// TIA Portal V17 export
// export: Created 2024-06-14T09:52:20.614085Z, ExportSetting WithDefaults, DisplayName Totally Integrated Automation Portal, DisplayVersion V17, DisplayName TIA Portal Openness, DisplayVersion V17, DisplayName TIA Portal Version Control Interface, DisplayVersion V17, DisplayName Simotion SCOUT TIA, DisplayVersion 5.4.3.0, DisplayName SINAMICS Startdrive Advanced, DisplayVersion V17 SP1 Update 1, DisplayName SINAMICS Startdrive G110M, G120, G120C, G120D, G120P, G115D, DisplayVersion V17 SP1 Update 1, DisplayName SINAMICS Startdrive G130, G150, S120, S150, SINAMICS MV, S210, DisplayVersion V17 SP1 Update 1, DisplayName STEP 7 Professional, DisplayVersion V17, DisplayName STEP 7 Safety, DisplayVersion V17, DisplayName WinCC Professional, DisplayVersion V17
FUNCTION_BLOCK "FILLING_FB_L2"   // FB12, LAD
{ S7_Optimized_Access := 'TRUE' }
VERSION : 0.1
// stored: AutoNumber false, IsIECCheckEnabled false, IsRetainMemResEnabled false, MemoryReserve 100, SetENOAutomatically false, UDAEnableTagReadback false
   VAR_INPUT
      CYCLE_START : Bool;
      CYCLE_RESET : Bool;
      CYL_STOPPER : Bool;
      CYL_SENSOR1 : Bool;
      CYL_SENSOR2 : Bool;
      CYL_SENSOR3 : Bool;
      CYL_SENSOR4 : Bool;
      CYL_SENSOR5 : Bool;
      CYL_SENSOR6 : Bool;
      "DOWN CONVEYOR" : Bool;
      "SENSING TIME" : DInt;
      ENABLE_CYLINDER { ExternalAccessible := 'False'; ExternalVisible := 'False'; ExternalWritable := 'False'} : Array[1..6] of Bool;
      ENABLED_CYLINDER { ExternalAccessible := 'False'; ExternalVisible := 'False'; ExternalWritable := 'False'} : Int;
      GUN_DELAY_TIME : DInt;
      FILL_SEQ_STARTED : Array[1..6] of Bool;
      FILLING_DONE : Array[1..6] of Bool;
   END_VAR
   VAR_OUTPUT
      STOPPER : Bool;
      "LIFT TABLE1" : Bool;
      "LIFT TABLE2" : Bool;
      "LIFT TABLE3" : Bool;
      "LIFT TABLE4" : Bool;
      "LIFT TABLE5" : Bool;
      "LIFT TABLE6" : Bool;
      GUN_DOWN1 : Bool;
      GUN_DOWN2 : Bool;
      GUN_DOWN3 : Bool;
      GUN_DOWN4 : Bool;
      GUN_DOWN5 : Bool;
      GUN_DOWN6 : Bool;
      CYCLE_RUNNING : Bool;
      FILL_STT_SEQ1 : Bool;
      FILL_STT_SEQ2 : Bool;
      FILL_STT_SEQ3 : Bool;
      FILL_STT_SEQ4 : Bool;
      FILL_STT_SEQ5 : Bool;
      FILL_STT_SEQ6 : Bool;
      FILLING_SEQ_DONE : Bool;
      ALL_STATION_DISABLED : Bool;
   END_VAR
   VAR
      "FIRST SCAN BIT" : Bool;
      CYCLE_OK : Bool;
      CYCLE_RESTART : Bool;
      "COUNTER RESET" : Bool;
      FIRST_CYCLE : Bool;
      "CYL COUNT  VALUE" : Int;
      "PLUS BIT" : Array[1..50] of Bool;
      "GUN DOWN" : Bool;
   END_VAR
   VAR RETAIN
      TILLTING_TIME { S7_SetPoint := 'True'} : DInt;
      M1_DECLAMP_TIME : DInt;
      CYL_COUNTER_S1 { S7_SetPoint := 'True'} : CTU_INT;
      CYL_COUNTER_S2 { S7_SetPoint := 'True'} : CTU_INT;
      CYL_COUNTER_S3 { S7_SetPoint := 'True'} : CTU_INT;
      CYL_COUNTER_S4 { S7_SetPoint := 'True'} : CTU_INT;
      CYL_COUNTER_S5 { S7_SetPoint := 'True'} : CTU_INT;
      CYL_COUNTER_S6 { S7_SetPoint := 'True'} : CTU_INT;
      CYL_COUNTER_S11 { S7_SetPoint := 'True'} : CTU_INT;
      CYL_COUNT_CONT_S1 { S7_SetPoint := 'True'} : CTU_INT;
      CYL_COUNT_CONT_S2 { S7_SetPoint := 'True'} : CTU_INT;
      CYL_COUNT_CONT_S3 { S7_SetPoint := 'True'} : CTU_INT;
      CYL_COUNT_CONT_S4 { S7_SetPoint := 'True'} : CTU_INT;
      CYL_COUNT_CONT_S5 { S7_SetPoint := 'True'} : CTU_INT;
      CYL_COUNT_CONT_S6 { S7_SetPoint := 'True'} : CTU_INT;
      "STOPPER COUNTER" { S7_SetPoint := 'True'} : CTU_INT;
   END_VAR
   VAR
      CYL_STAB_S1 { S7_SetPoint := 'True'} : TON_TIME;
      CYL_STAB_S2 { S7_SetPoint := 'True'} : TON_TIME;
      CYL_STAB_S3 { S7_SetPoint := 'True'} : TON_TIME;
      CYL_STAB_S4 { S7_SetPoint := 'True'} : TON_TIME;
      CYL_STAB_S5 { S7_SetPoint := 'True'} : TON_TIME;
      CYL_STAB_S6 { S7_SetPoint := 'True'} : TON_TIME;
      CYCLE_RST_OFF { S7_SetPoint := 'True'} : TOF_TIME;
      CYCLE_RST_ON { S7_SetPoint := 'True'} : TON_TIME;
      DECLAMP_MUL : DInt;
      DECLAMP_ADD : DInt;
      "CYL STOPPER" : Bool;
      STOP_DLY { S7_SetPoint := 'True'} : TON_TIME;
      Disable_Stations { S7_SetPoint := 'True'} : "Disable";
      First_Cylinder : Array[1..6] of Int;
      Disab_Total_Cyl : Int;
      GUN_DOWN_FBK : Bool;
      GUN_DOWN_FBK_T { S7_SetPoint := 'True'} : TON_TIME;
      AUTO_RESTART : Bool;
      GUN_DOWN_1 { S7_SetPoint := 'True'} : TON_TIME;
      GUN_DOWN_2 { S7_SetPoint := 'True'} : TON_TIME;
      GUN_DOWN_3 { S7_SetPoint := 'True'} : TON_TIME;
      GUN_DOWN_4 { S7_SetPoint := 'True'} : TON_TIME;
      GUN_DOWN_5 { S7_SetPoint := 'True'} : TON_TIME;
      GUN_DOWN_6 { S7_SetPoint := 'True'} : TON_TIME;
      FILL_STT_1 { S7_SetPoint := 'True'} : TON_TIME;
      FILL_STT_2 { S7_SetPoint := 'True'} : TON_TIME;
      FILL_STT_3 { S7_SetPoint := 'True'} : TON_TIME;
      FILL_STT_4 { S7_SetPoint := 'True'} : TON_TIME;
      FILL_STT_5 { S7_SetPoint := 'True'} : TON_TIME;
      FILL_STT_6 { S7_SetPoint := 'True'} : TON_TIME;
      ALL_FILL_DONE : Bool;
      ALL_GUN_UP : Bool;
      AUTO_CYCLE { S7_SetPoint := 'True'} : TON_TIME;
      AUTO { S7_SetPoint := 'True'} : Bool;
      MANUAL { S7_SetPoint := 'True'} : Bool;
      Man_Gun_down_1 : Bool;
      Man_Gun_down_2 : Bool;
      Man_Gun_down_3 : Bool;
      Man_Gun_down_4 : Bool;
      Man_Gun_down_5 : Bool;
      Man_Gun_down_6 : Bool;
      Man_Lift_up_1 : Bool;
      Man_Lift_up_2 : Bool;
      Man_Lift_up_3 : Bool;
      Man_Lift_up_4 : Bool;
      Man_Lift_up_5 : Bool;
      Man_Lift_up_6 : Bool;
      trig : Array[0..50] of Bool;
      "trig count" : Array[0..10] of TON_TIME;
      delay : Time;
   END_VAR
   VAR_TEMP   // added for the SCL form of the ladder/FBD networks
      _w1 : Bool;
      _w2 : Bool;
      _w3 : Bool;
      _w4 : Bool;
      _w5 : Bool;
      _w6 : Bool;
      _w7 : Bool;
      _w8 : Bool;
      _w9 : Bool;
      _w10 : Bool;
      _w11 : Bool;
      _w12 : Bool;
      _w13 : Bool;
      _w14 : Bool;
      _w15 : Bool;
      _w16 : Bool;
      _w17 : Bool;
      _w18 : Bool;
      _w19 : Bool;
      _w20 : Bool;
      _w21 : Bool;
      _w22 : Bool;
      _w23 : Bool;
      _w24 : Bool;
      _w25 : Bool;
      _w26 : Bool;
      _w27 : Bool;
      _w28 : Bool;
      _w29 : Bool;
      _w30 : Bool;
      _w31 : Bool;
   END_VAR
BEGIN

REGION Network 2: CYCLE START / POWER RESET OFF
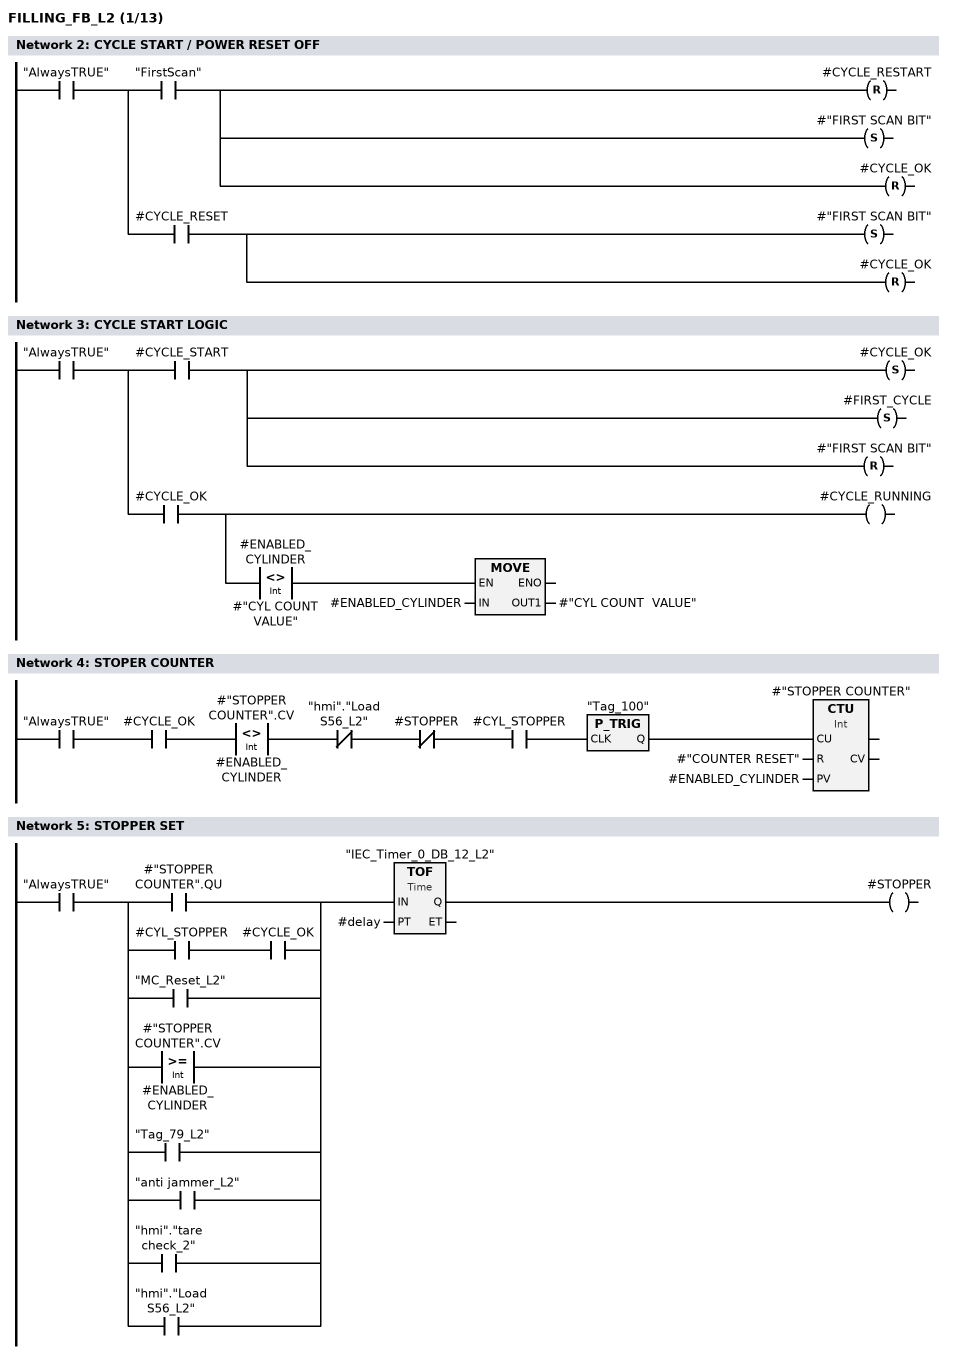
   RUNG wire#powerrail
      Contact( "AlwaysTRUE" )
      wire#w1
      Contact( "FirstScan" )
      wire#w2
      R_Coil( #CYCLE_RESTART )
   END_RUNG
   RUNG wire#w2
      S_Coil( #"FIRST SCAN BIT" )
   END_RUNG
   RUNG wire#w2
      R_Coil( #CYCLE_OK )
   END_RUNG
   RUNG wire#w1
      Contact( #CYCLE_RESET )
      wire#w3
      S_Coil( #"FIRST SCAN BIT" )
   END_RUNG
   RUNG wire#w3
      R_Coil( #CYCLE_OK )
   END_RUNG
   // the same network as SCL:
   IF "AlwaysTRUE" AND "FirstScan" THEN
       #CYCLE_RESTART := FALSE;
       #"FIRST SCAN BIT" := TRUE;
       #CYCLE_OK := FALSE;
   END_IF;
   IF "AlwaysTRUE" AND #CYCLE_RESET THEN
       #"FIRST SCAN BIT" := TRUE;
       #CYCLE_OK := FALSE;
   END_IF;
END_REGION

REGION Network 3: CYCLE START LOGIC
   RUNG wire#powerrail
      Contact( "AlwaysTRUE" )
      wire#w1
      Contact( #CYCLE_START )
      wire#w2
      S_Coil( #CYCLE_OK )
   END_RUNG
   RUNG wire#w2
      S_Coil( #FIRST_CYCLE )
   END_RUNG
   RUNG wire#w2
      R_Coil( #"FIRST SCAN BIT" )
   END_RUNG
   RUNG wire#w1
      Contact( #CYCLE_OK )
      wire#w3
      Coil( #CYCLE_RUNNING )
   END_RUNG
   RUNG wire#w3
      { S7_Templates := "SrcType := Int" } NE_Contact(in1 := #ENABLED_CYLINDER, in2 := #"CYL COUNT  VALUE")
      Move(in := #ENABLED_CYLINDER, out1 => #"CYL COUNT  VALUE")
   END_RUNG
   // the same network as SCL:
   IF "AlwaysTRUE" AND #CYCLE_START THEN
       #CYCLE_OK := TRUE;
       #FIRST_CYCLE := TRUE;
       #"FIRST SCAN BIT" := FALSE;
   END_IF;
   #CYCLE_RUNNING := "AlwaysTRUE" AND #CYCLE_OK;
   IF #CYCLE_RUNNING AND (#ENABLED_CYLINDER <> #"CYL COUNT  VALUE") THEN
       #"CYL COUNT  VALUE" := #ENABLED_CYLINDER;
   END_IF;
END_REGION

REGION Network 4: STOPER COUNTER
   RUNG wire#powerrail
      Contact( "AlwaysTRUE" )
      Contact( #CYCLE_OK )
      { S7_Templates := "SrcType := Int" } NE_Contact(in1 := #"STOPPER COUNTER".CV, in2 := #ENABLED_CYLINDER)
      I_Contact( "hmi"."Load S56_L2" )
      I_Contact( #STOPPER )
      Contact( #CYL_STOPPER )
      P_Trig( "Tag_100" )
      { S7_Templates := "value_type := Int" } #"STOPPER COUNTER".CTU(r := #"COUNTER RESET", pv := #ENABLED_CYLINDER, cv =>)
   END_RUNG
   // the same network as SCL:
   #_w1 := "AlwaysTRUE" AND #CYCLE_OK AND (#"STOPPER COUNTER".CV <> #ENABLED_CYLINDER) AND NOT "hmi"."Load S56_L2" AND NOT #STOPPER AND #CYL_STOPPER;
   #_w2 := #_w1 AND NOT "Tag_100";   // rising edge
   "Tag_100" := #_w1;
   #"STOPPER COUNTER"(CU := #_w2, R := #"COUNTER RESET", PV := #ENABLED_CYLINDER);   // CTU
END_REGION

REGION Network 5: STOPPER SET
   RUNG wire#powerrail
      Contact( "AlwaysTRUE" )
      wire#w1
      Contact( #"STOPPER COUNTER".QU )
      wire#w2
      { S7_Templates := "time_type := Time" } "IEC_Timer_0_DB_12_L2".TOF(pt := #delay, et =>)
      Coil( #STOPPER )
   END_RUNG
   RUNG wire#w1
      Contact( #CYL_STOPPER )
      Contact( #CYCLE_OK )
   END_RUNG wire#w2
   RUNG wire#w1
      Contact( "MC_Reset_L2" )
   END_RUNG wire#w2
   RUNG wire#w1
      { S7_Templates := "SrcType := Int" } GE_Contact(in1 := #"STOPPER COUNTER".CV, in2 := #ENABLED_CYLINDER)
   END_RUNG wire#w2
   RUNG wire#w1
      Contact( "Tag_79_L2" )
   END_RUNG wire#w2
   RUNG wire#w1
      Contact( "anti jammer_L2" )
   END_RUNG wire#w2
   RUNG wire#w1
      Contact( "hmi"."tare check_2" )
   END_RUNG wire#w2
   RUNG wire#w1
      Contact( "hmi"."Load S56_L2" )
   END_RUNG wire#w2
   // the same network as SCL:
   "IEC_Timer_0_DB_12_L2".TOF(IN := "AlwaysTRUE" AND (#"STOPPER COUNTER".QU OR (#CYL_STOPPER AND #CYCLE_OK) OR "MC_Reset_L2" OR (#"STOPPER COUNTER".CV >= #ENABLED_CYLINDER) OR "Tag_79_L2" OR "anti jammer_L2" OR "hmi"."tare check_2" OR "hmi"."Load S56_L2"),
                           PT := #delay);
   #STOPPER := "IEC_Timer_0_DB_12_L2".Q;
END_REGION

REGION Network 6
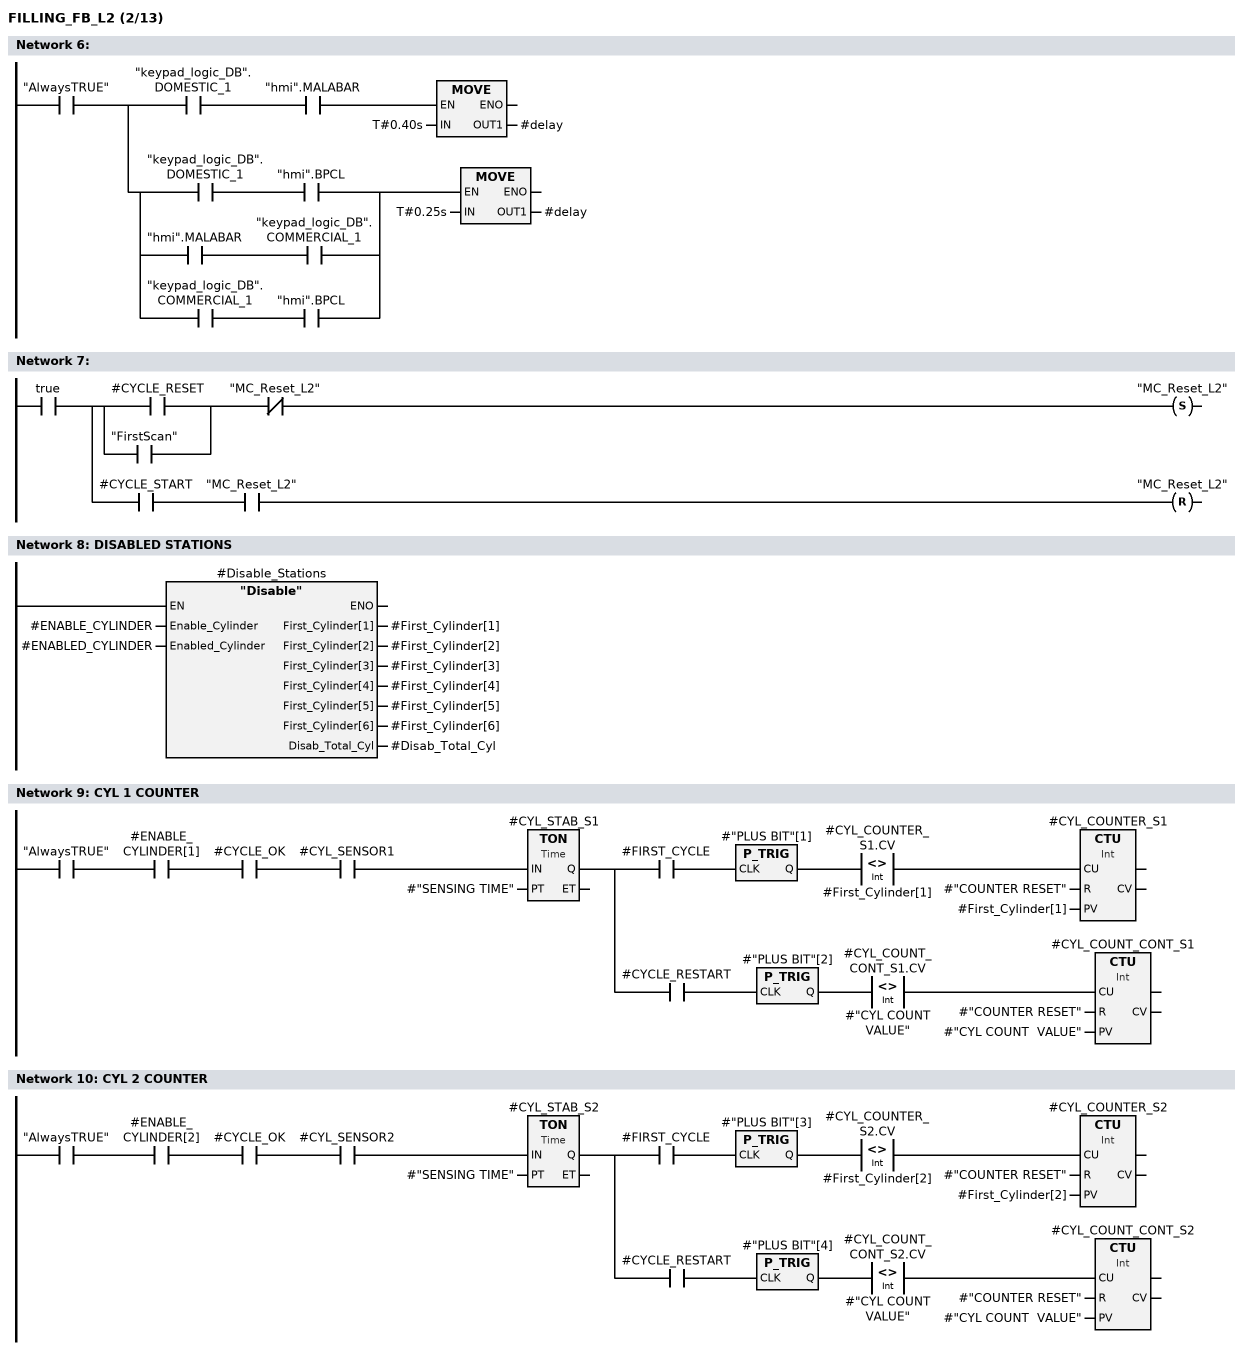
   RUNG wire#powerrail
      Contact( "AlwaysTRUE" )
      wire#w1
      Contact( "keypad_logic_DB".DOMESTIC_1 )
      Contact( "hmi".MALABAR )
      Move(in := T#0.40s, out1 => #delay)
   END_RUNG
   RUNG wire#w1
      Contact( "keypad_logic_DB".DOMESTIC_1 )
      Contact( "hmi".BPCL )
      wire#w2
      Move(in := T#0.25s, out1 => #delay)
   END_RUNG
   RUNG wire#w1
      Contact( "hmi".MALABAR )
      Contact( "keypad_logic_DB".COMMERCIAL_1 )
   END_RUNG wire#w2
   RUNG wire#w1
      Contact( "keypad_logic_DB".COMMERCIAL_1 )
      Contact( "hmi".BPCL )
   END_RUNG wire#w2
   // the same network as SCL:
   IF "AlwaysTRUE" AND "keypad_logic_DB".DOMESTIC_1 AND "hmi".MALABAR THEN #delay := T#0.40s; END_IF;
   IF "AlwaysTRUE" AND (("keypad_logic_DB".DOMESTIC_1 AND "hmi".BPCL) OR ("hmi".MALABAR AND "keypad_logic_DB".COMMERCIAL_1) OR ("keypad_logic_DB".COMMERCIAL_1 AND "hmi".BPCL)) THEN
       #delay := T#0.25s;
   END_IF;
END_REGION

REGION Network 7
   RUNG wire#powerrail
      Contact( true )
      wire#w1
      Contact( #CYCLE_RESET )
      wire#w2
      I_Contact( "MC_Reset_L2" )
      S_Coil( "MC_Reset_L2" )
   END_RUNG
   RUNG wire#w1
      Contact( "FirstScan" )
   END_RUNG wire#w2
   RUNG wire#w1
      Contact( #CYCLE_START )
      Contact( "MC_Reset_L2" )
      R_Coil( "MC_Reset_L2" )
   END_RUNG
   // the same network as SCL:
   IF true AND (#CYCLE_RESET OR "FirstScan") AND NOT "MC_Reset_L2" THEN "MC_Reset_L2" := TRUE; END_IF;
   IF true AND #CYCLE_START AND "MC_Reset_L2" THEN "MC_Reset_L2" := FALSE; END_IF;
END_REGION

REGION Network 8: DISABLED STATIONS
   RUNG wire#powerrail
      #Disable_Stations(Enable_Cylinder := #ENABLE_CYLINDER, Enabled_Cylinder := #ENABLED_CYLINDER, "First_Cylinder[1]" => #First_Cylinder[1], "First_Cylinder[2]" => #First_Cylinder[2], "First_Cylinder[3]" => #First_Cylinder[3], "First_Cylinder[4]" => #First_Cylinder[4], "First_Cylinder[5]" => #First_Cylinder[5], "First_Cylinder[6]" => #First_Cylinder[6], Disab_Total_Cyl => #Disab_Total_Cyl)
   END_RUNG
   // the same network as SCL:
   #Disable_Stations(Enable_Cylinder := #ENABLE_CYLINDER,   // "Disable"
                     Enabled_Cylinder := #ENABLED_CYLINDER,
                     "First_Cylinder[1]" => #First_Cylinder[1],
                     "First_Cylinder[2]" => #First_Cylinder[2],
                     "First_Cylinder[3]" => #First_Cylinder[3],
                     "First_Cylinder[4]" => #First_Cylinder[4],
                     "First_Cylinder[5]" => #First_Cylinder[5],
                     "First_Cylinder[6]" => #First_Cylinder[6],
                     Disab_Total_Cyl => #Disab_Total_Cyl);
END_REGION

REGION Network 9: CYL 1 COUNTER
   RUNG wire#powerrail
      Contact( "AlwaysTRUE" )
      Contact( #ENABLE_CYLINDER[1] )
      Contact( #CYCLE_OK )
      Contact( #CYL_SENSOR1 )
      { S7_Templates := "time_type := Time" } #CYL_STAB_S1.TON(pt := #"SENSING TIME", et =>)
      wire#w1
      Contact( #FIRST_CYCLE )
      P_Trig( #"PLUS BIT"[1] )
      { S7_Templates := "SrcType := Int" } NE_Contact(in1 := #CYL_COUNTER_S1.CV, in2 := #First_Cylinder[1])
      { S7_Templates := "value_type := Int" } #CYL_COUNTER_S1.CTU(r := #"COUNTER RESET", pv := #First_Cylinder[1], cv =>)
   END_RUNG
   RUNG wire#w1
      Contact( #CYCLE_RESTART )
      P_Trig( #"PLUS BIT"[2] )
      { S7_Templates := "SrcType := Int" } NE_Contact(in1 := #CYL_COUNT_CONT_S1.CV, in2 := #"CYL COUNT  VALUE")
      { S7_Templates := "value_type := Int" } #CYL_COUNT_CONT_S1.CTU(r := #"COUNTER RESET", pv := #"CYL COUNT  VALUE", cv =>)
   END_RUNG
   // the same network as SCL:
   #CYL_STAB_S1(IN := "AlwaysTRUE" AND #ENABLE_CYLINDER[1] AND #CYCLE_OK AND #CYL_SENSOR1,   // TON
                PT := #"SENSING TIME");
   #_w1 := #CYL_STAB_S1.Q AND #FIRST_CYCLE;
   #_w2 := #_w1 AND NOT #"PLUS BIT"[1];   // rising edge
   #"PLUS BIT"[1] := #_w1;
   #CYL_COUNTER_S1(CU := #_w2 AND (#CYL_COUNTER_S1.CV <> #First_Cylinder[1]),   // CTU
                   R := #"COUNTER RESET",
                   PV := #First_Cylinder[1]);
   #_w3 := #CYL_STAB_S1.Q AND #CYCLE_RESTART;
   #_w4 := #_w3 AND NOT #"PLUS BIT"[2];   // rising edge
   #"PLUS BIT"[2] := #_w3;
   #CYL_COUNT_CONT_S1(CU := #_w4 AND (#CYL_COUNT_CONT_S1.CV <> #"CYL COUNT  VALUE"),   // CTU
                      R := #"COUNTER RESET",
                      PV := #"CYL COUNT  VALUE");
END_REGION

REGION Network 10: CYL 2 COUNTER
   RUNG wire#powerrail
      Contact( "AlwaysTRUE" )
      Contact( #ENABLE_CYLINDER[2] )
      Contact( #CYCLE_OK )
      Contact( #CYL_SENSOR2 )
      { S7_Templates := "time_type := Time" } #CYL_STAB_S2.TON(pt := #"SENSING TIME", et =>)
      wire#w1
      Contact( #FIRST_CYCLE )
      P_Trig( #"PLUS BIT"[3] )
      { S7_Templates := "SrcType := Int" } NE_Contact(in1 := #CYL_COUNTER_S2.CV, in2 := #First_Cylinder[2])
      { S7_Templates := "value_type := Int" } #CYL_COUNTER_S2.CTU(r := #"COUNTER RESET", pv := #First_Cylinder[2], cv =>)
   END_RUNG
   RUNG wire#w1
      Contact( #CYCLE_RESTART )
      P_Trig( #"PLUS BIT"[4] )
      { S7_Templates := "SrcType := Int" } NE_Contact(in1 := #CYL_COUNT_CONT_S2.CV, in2 := #"CYL COUNT  VALUE")
      { S7_Templates := "value_type := Int" } #CYL_COUNT_CONT_S2.CTU(r := #"COUNTER RESET", pv := #"CYL COUNT  VALUE", cv =>)
   END_RUNG
   // the same network as SCL:
   #CYL_STAB_S2(IN := "AlwaysTRUE" AND #ENABLE_CYLINDER[2] AND #CYCLE_OK AND #CYL_SENSOR2,   // TON
                PT := #"SENSING TIME");
   #_w1 := #CYL_STAB_S2.Q AND #FIRST_CYCLE;
   #_w2 := #_w1 AND NOT #"PLUS BIT"[3];   // rising edge
   #"PLUS BIT"[3] := #_w1;
   #CYL_COUNTER_S2(CU := #_w2 AND (#CYL_COUNTER_S2.CV <> #First_Cylinder[2]),   // CTU
                   R := #"COUNTER RESET",
                   PV := #First_Cylinder[2]);
   #_w3 := #CYL_STAB_S2.Q AND #CYCLE_RESTART;
   #_w4 := #_w3 AND NOT #"PLUS BIT"[4];   // rising edge
   #"PLUS BIT"[4] := #_w3;
   #CYL_COUNT_CONT_S2(CU := #_w4 AND (#CYL_COUNT_CONT_S2.CV <> #"CYL COUNT  VALUE"),   // CTU
                      R := #"COUNTER RESET",
                      PV := #"CYL COUNT  VALUE");
END_REGION

REGION Network 11: CYL 3 COUNTER
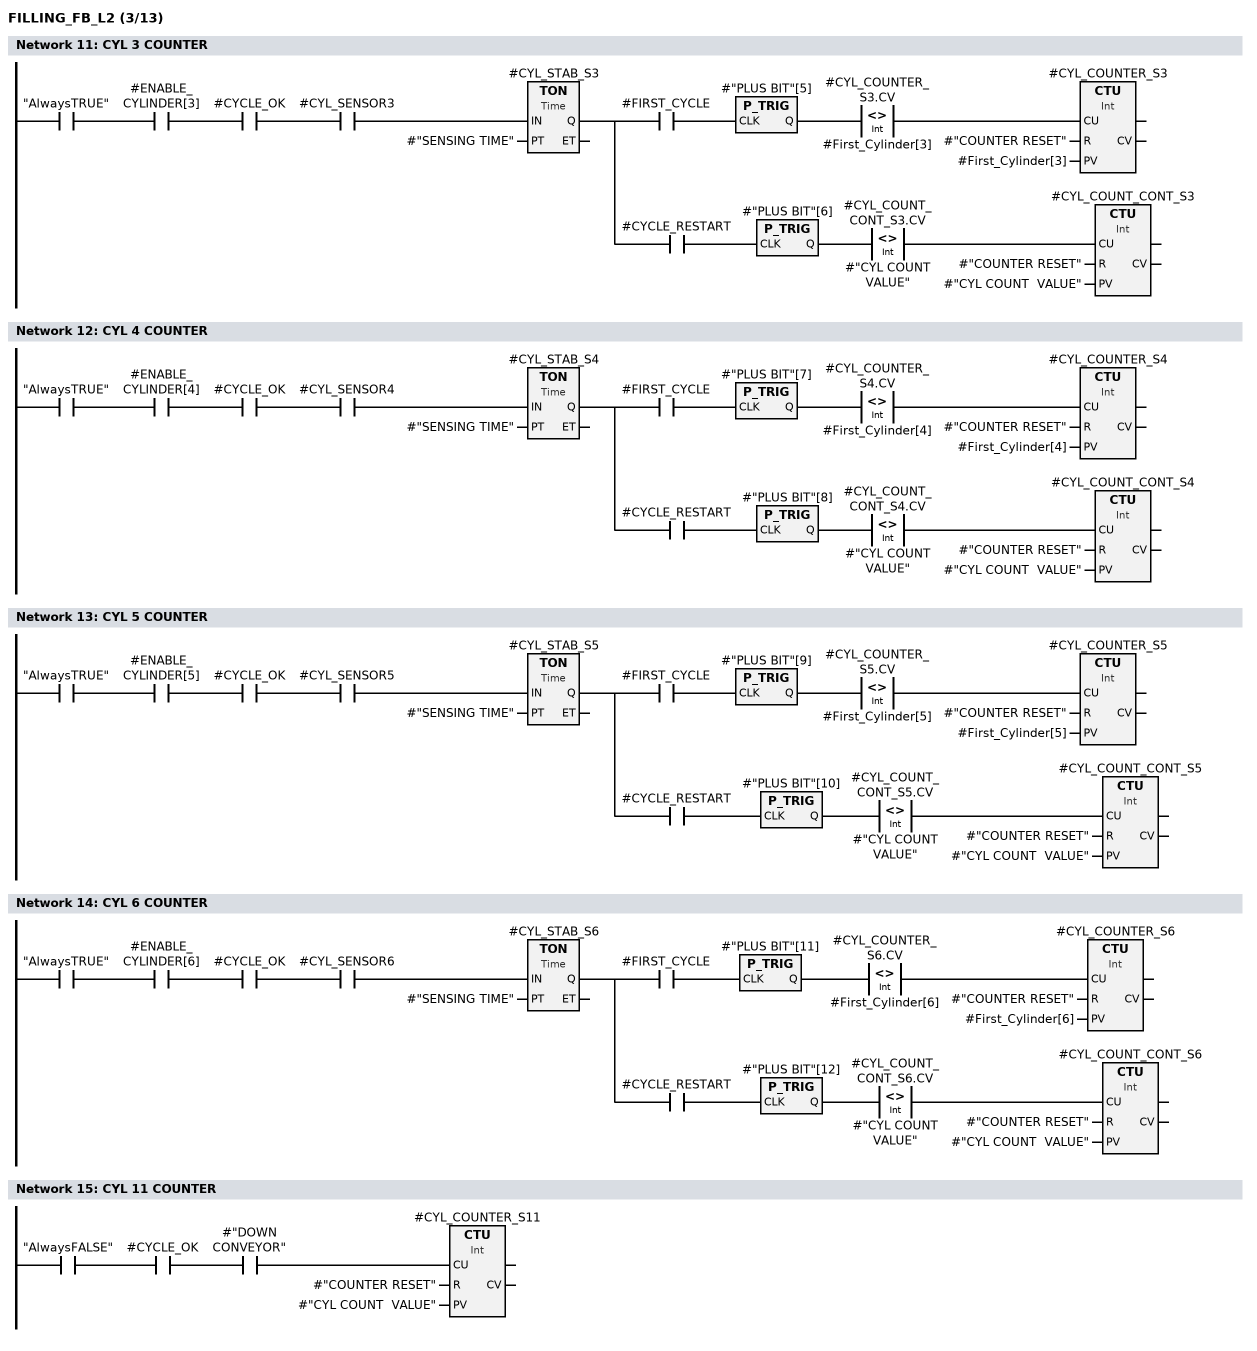
   RUNG wire#powerrail
      Contact( "AlwaysTRUE" )
      Contact( #ENABLE_CYLINDER[3] )
      Contact( #CYCLE_OK )
      Contact( #CYL_SENSOR3 )
      { S7_Templates := "time_type := Time" } #CYL_STAB_S3.TON(pt := #"SENSING TIME", et =>)
      wire#w1
      Contact( #FIRST_CYCLE )
      P_Trig( #"PLUS BIT"[5] )
      { S7_Templates := "SrcType := Int" } NE_Contact(in1 := #CYL_COUNTER_S3.CV, in2 := #First_Cylinder[3])
      { S7_Templates := "value_type := Int" } #CYL_COUNTER_S3.CTU(r := #"COUNTER RESET", pv := #First_Cylinder[3], cv =>)
   END_RUNG
   RUNG wire#w1
      Contact( #CYCLE_RESTART )
      P_Trig( #"PLUS BIT"[6] )
      { S7_Templates := "SrcType := Int" } NE_Contact(in1 := #CYL_COUNT_CONT_S3.CV, in2 := #"CYL COUNT  VALUE")
      { S7_Templates := "value_type := Int" } #CYL_COUNT_CONT_S3.CTU(r := #"COUNTER RESET", pv := #"CYL COUNT  VALUE", cv =>)
   END_RUNG
   // the same network as SCL:
   #CYL_STAB_S3(IN := "AlwaysTRUE" AND #ENABLE_CYLINDER[3] AND #CYCLE_OK AND #CYL_SENSOR3,   // TON
                PT := #"SENSING TIME");
   #_w1 := #CYL_STAB_S3.Q AND #FIRST_CYCLE;
   #_w2 := #_w1 AND NOT #"PLUS BIT"[5];   // rising edge
   #"PLUS BIT"[5] := #_w1;
   #CYL_COUNTER_S3(CU := #_w2 AND (#CYL_COUNTER_S3.CV <> #First_Cylinder[3]),   // CTU
                   R := #"COUNTER RESET",
                   PV := #First_Cylinder[3]);
   #_w3 := #CYL_STAB_S3.Q AND #CYCLE_RESTART;
   #_w4 := #_w3 AND NOT #"PLUS BIT"[6];   // rising edge
   #"PLUS BIT"[6] := #_w3;
   #CYL_COUNT_CONT_S3(CU := #_w4 AND (#CYL_COUNT_CONT_S3.CV <> #"CYL COUNT  VALUE"),   // CTU
                      R := #"COUNTER RESET",
                      PV := #"CYL COUNT  VALUE");
END_REGION

REGION Network 12: CYL 4 COUNTER
   RUNG wire#powerrail
      Contact( "AlwaysTRUE" )
      Contact( #ENABLE_CYLINDER[4] )
      Contact( #CYCLE_OK )
      Contact( #CYL_SENSOR4 )
      { S7_Templates := "time_type := Time" } #CYL_STAB_S4.TON(pt := #"SENSING TIME", et =>)
      wire#w1
      Contact( #FIRST_CYCLE )
      P_Trig( #"PLUS BIT"[7] )
      { S7_Templates := "SrcType := Int" } NE_Contact(in1 := #CYL_COUNTER_S4.CV, in2 := #First_Cylinder[4])
      { S7_Templates := "value_type := Int" } #CYL_COUNTER_S4.CTU(r := #"COUNTER RESET", pv := #First_Cylinder[4], cv =>)
   END_RUNG
   RUNG wire#w1
      Contact( #CYCLE_RESTART )
      P_Trig( #"PLUS BIT"[8] )
      { S7_Templates := "SrcType := Int" } NE_Contact(in1 := #CYL_COUNT_CONT_S4.CV, in2 := #"CYL COUNT  VALUE")
      { S7_Templates := "value_type := Int" } #CYL_COUNT_CONT_S4.CTU(r := #"COUNTER RESET", pv := #"CYL COUNT  VALUE", cv =>)
   END_RUNG
   // the same network as SCL:
   #CYL_STAB_S4(IN := "AlwaysTRUE" AND #ENABLE_CYLINDER[4] AND #CYCLE_OK AND #CYL_SENSOR4,   // TON
                PT := #"SENSING TIME");
   #_w1 := #CYL_STAB_S4.Q AND #FIRST_CYCLE;
   #_w2 := #_w1 AND NOT #"PLUS BIT"[7];   // rising edge
   #"PLUS BIT"[7] := #_w1;
   #CYL_COUNTER_S4(CU := #_w2 AND (#CYL_COUNTER_S4.CV <> #First_Cylinder[4]),   // CTU
                   R := #"COUNTER RESET",
                   PV := #First_Cylinder[4]);
   #_w3 := #CYL_STAB_S4.Q AND #CYCLE_RESTART;
   #_w4 := #_w3 AND NOT #"PLUS BIT"[8];   // rising edge
   #"PLUS BIT"[8] := #_w3;
   #CYL_COUNT_CONT_S4(CU := #_w4 AND (#CYL_COUNT_CONT_S4.CV <> #"CYL COUNT  VALUE"),   // CTU
                      R := #"COUNTER RESET",
                      PV := #"CYL COUNT  VALUE");
END_REGION

REGION Network 13: CYL 5 COUNTER
   RUNG wire#powerrail
      Contact( "AlwaysTRUE" )
      Contact( #ENABLE_CYLINDER[5] )
      Contact( #CYCLE_OK )
      Contact( #CYL_SENSOR5 )
      { S7_Templates := "time_type := Time" } #CYL_STAB_S5.TON(pt := #"SENSING TIME", et =>)
      wire#w1
      Contact( #FIRST_CYCLE )
      P_Trig( #"PLUS BIT"[9] )
      { S7_Templates := "SrcType := Int" } NE_Contact(in1 := #CYL_COUNTER_S5.CV, in2 := #First_Cylinder[5])
      { S7_Templates := "value_type := Int" } #CYL_COUNTER_S5.CTU(r := #"COUNTER RESET", pv := #First_Cylinder[5], cv =>)
   END_RUNG
   RUNG wire#w1
      Contact( #CYCLE_RESTART )
      P_Trig( #"PLUS BIT"[10] )
      { S7_Templates := "SrcType := Int" } NE_Contact(in1 := #CYL_COUNT_CONT_S5.CV, in2 := #"CYL COUNT  VALUE")
      { S7_Templates := "value_type := Int" } #CYL_COUNT_CONT_S5.CTU(r := #"COUNTER RESET", pv := #"CYL COUNT  VALUE", cv =>)
   END_RUNG
   // the same network as SCL:
   #CYL_STAB_S5(IN := "AlwaysTRUE" AND #ENABLE_CYLINDER[5] AND #CYCLE_OK AND #CYL_SENSOR5,   // TON
                PT := #"SENSING TIME");
   #_w1 := #CYL_STAB_S5.Q AND #FIRST_CYCLE;
   #_w2 := #_w1 AND NOT #"PLUS BIT"[9];   // rising edge
   #"PLUS BIT"[9] := #_w1;
   #CYL_COUNTER_S5(CU := #_w2 AND (#CYL_COUNTER_S5.CV <> #First_Cylinder[5]),   // CTU
                   R := #"COUNTER RESET",
                   PV := #First_Cylinder[5]);
   #_w3 := #CYL_STAB_S5.Q AND #CYCLE_RESTART;
   #_w4 := #_w3 AND NOT #"PLUS BIT"[10];   // rising edge
   #"PLUS BIT"[10] := #_w3;
   #CYL_COUNT_CONT_S5(CU := #_w4 AND (#CYL_COUNT_CONT_S5.CV <> #"CYL COUNT  VALUE"),   // CTU
                      R := #"COUNTER RESET",
                      PV := #"CYL COUNT  VALUE");
END_REGION

REGION Network 14: CYL 6 COUNTER
   RUNG wire#powerrail
      Contact( "AlwaysTRUE" )
      Contact( #ENABLE_CYLINDER[6] )
      Contact( #CYCLE_OK )
      Contact( #CYL_SENSOR6 )
      { S7_Templates := "time_type := Time" } #CYL_STAB_S6.TON(pt := #"SENSING TIME", et =>)
      wire#w1
      Contact( #FIRST_CYCLE )
      P_Trig( #"PLUS BIT"[11] )
      { S7_Templates := "SrcType := Int" } NE_Contact(in1 := #CYL_COUNTER_S6.CV, in2 := #First_Cylinder[6])
      { S7_Templates := "value_type := Int" } #CYL_COUNTER_S6.CTU(r := #"COUNTER RESET", pv := #First_Cylinder[6], cv =>)
   END_RUNG
   RUNG wire#w1
      Contact( #CYCLE_RESTART )
      P_Trig( #"PLUS BIT"[12] )
      { S7_Templates := "SrcType := Int" } NE_Contact(in1 := #CYL_COUNT_CONT_S6.CV, in2 := #"CYL COUNT  VALUE")
      { S7_Templates := "value_type := Int" } #CYL_COUNT_CONT_S6.CTU(r := #"COUNTER RESET", pv := #"CYL COUNT  VALUE", cv =>)
   END_RUNG
   // the same network as SCL:
   #CYL_STAB_S6(IN := "AlwaysTRUE" AND #ENABLE_CYLINDER[6] AND #CYCLE_OK AND #CYL_SENSOR6,   // TON
                PT := #"SENSING TIME");
   #_w1 := #CYL_STAB_S6.Q AND #FIRST_CYCLE;
   #_w2 := #_w1 AND NOT #"PLUS BIT"[11];   // rising edge
   #"PLUS BIT"[11] := #_w1;
   #CYL_COUNTER_S6(CU := #_w2 AND (#CYL_COUNTER_S6.CV <> #First_Cylinder[6]),   // CTU
                   R := #"COUNTER RESET",
                   PV := #First_Cylinder[6]);
   #_w3 := #CYL_STAB_S6.Q AND #CYCLE_RESTART;
   #_w4 := #_w3 AND NOT #"PLUS BIT"[12];   // rising edge
   #"PLUS BIT"[12] := #_w3;
   #CYL_COUNT_CONT_S6(CU := #_w4 AND (#CYL_COUNT_CONT_S6.CV <> #"CYL COUNT  VALUE"),   // CTU
                      R := #"COUNTER RESET",
                      PV := #"CYL COUNT  VALUE");
END_REGION

REGION Network 15: CYL 11 COUNTER
   RUNG wire#powerrail
      Contact( "AlwaysFALSE" )
      Contact( #CYCLE_OK )
      Contact( #"DOWN CONVEYOR" )
      { S7_Templates := "value_type := Int" } #CYL_COUNTER_S11.CTU(r := #"COUNTER RESET", pv := #"CYL COUNT  VALUE", cv =>)
   END_RUNG
   // the same network as SCL:
   #CYL_COUNTER_S11(CU := "AlwaysFALSE" AND #CYCLE_OK AND #"DOWN CONVEYOR",   // CTU
                    R := #"COUNTER RESET",
                    PV := #"CYL COUNT  VALUE");
END_REGION

REGION Network 16: CYL 1 LOCK
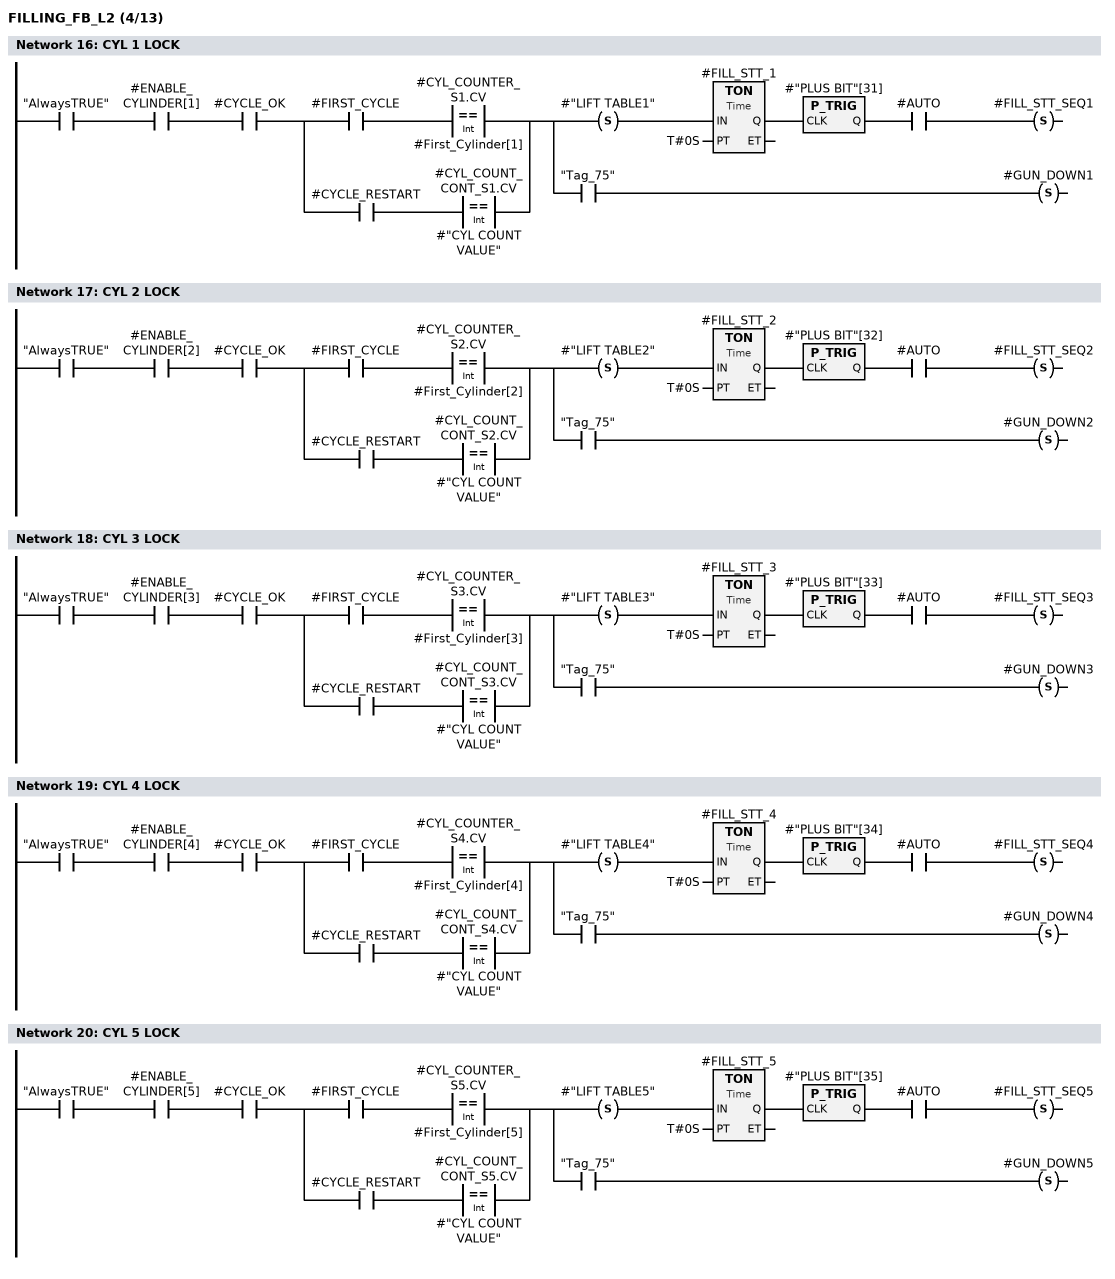
   RUNG wire#powerrail
      Contact( "AlwaysTRUE" )
      Contact( #ENABLE_CYLINDER[1] )
      Contact( #CYCLE_OK )
      wire#w1
      Contact( #FIRST_CYCLE )
      { S7_Templates := "SrcType := Int" } EQ_Contact(in1 := #CYL_COUNTER_S1.CV, in2 := #First_Cylinder[1])
      wire#w2
      S_Coil( #"LIFT TABLE1" )
      { S7_Templates := "time_type := Time" } #FILL_STT_1.TON(pt := T#0S, et =>)
      P_Trig( #"PLUS BIT"[31] )
      Contact( #AUTO )
      S_Coil( #FILL_STT_SEQ1 )
   END_RUNG
   RUNG wire#w1
      Contact( #CYCLE_RESTART )
      { S7_Templates := "SrcType := Int" } EQ_Contact(in1 := #CYL_COUNT_CONT_S1.CV, in2 := #"CYL COUNT  VALUE")
   END_RUNG wire#w2
   RUNG wire#w2
      Contact( "Tag_75" )
      S_Coil( #GUN_DOWN1 )
   END_RUNG
   // the same network as SCL:
   #_w1 := "AlwaysTRUE" AND #ENABLE_CYLINDER[1] AND #CYCLE_OK AND ((#FIRST_CYCLE AND (#CYL_COUNTER_S1.CV = #First_Cylinder[1])) OR (#CYCLE_RESTART AND (#CYL_COUNT_CONT_S1.CV = #"CYL COUNT  VALUE")));
   IF #_w1 THEN #"LIFT TABLE1" := TRUE; END_IF;
   #FILL_STT_1(IN := #_w1, PT := T#0S);   // TON
   #_w2 := #FILL_STT_1.Q AND NOT #"PLUS BIT"[31];   // rising edge
   #"PLUS BIT"[31] := #FILL_STT_1.Q;
   IF #_w2 AND #AUTO THEN #FILL_STT_SEQ1 := TRUE; END_IF;
   IF #_w1 AND "Tag_75" THEN #GUN_DOWN1 := TRUE; END_IF;
END_REGION

REGION Network 17: CYL 2 LOCK
   RUNG wire#powerrail
      Contact( "AlwaysTRUE" )
      Contact( #ENABLE_CYLINDER[2] )
      Contact( #CYCLE_OK )
      wire#w1
      Contact( #FIRST_CYCLE )
      { S7_Templates := "SrcType := Int" } EQ_Contact(in1 := #CYL_COUNTER_S2.CV, in2 := #First_Cylinder[2])
      wire#w2
      S_Coil( #"LIFT TABLE2" )
      { S7_Templates := "time_type := Time" } #FILL_STT_2.TON(pt := T#0S, et =>)
      P_Trig( #"PLUS BIT"[32] )
      Contact( #AUTO )
      S_Coil( #FILL_STT_SEQ2 )
   END_RUNG
   RUNG wire#w1
      Contact( #CYCLE_RESTART )
      { S7_Templates := "SrcType := Int" } EQ_Contact(in1 := #CYL_COUNT_CONT_S2.CV, in2 := #"CYL COUNT  VALUE")
   END_RUNG wire#w2
   RUNG wire#w2
      Contact( "Tag_75" )
      S_Coil( #GUN_DOWN2 )
   END_RUNG
   // the same network as SCL:
   #_w1 := "AlwaysTRUE" AND #ENABLE_CYLINDER[2] AND #CYCLE_OK AND ((#FIRST_CYCLE AND (#CYL_COUNTER_S2.CV = #First_Cylinder[2])) OR (#CYCLE_RESTART AND (#CYL_COUNT_CONT_S2.CV = #"CYL COUNT  VALUE")));
   IF #_w1 THEN #"LIFT TABLE2" := TRUE; END_IF;
   #FILL_STT_2(IN := #_w1, PT := T#0S);   // TON
   #_w2 := #FILL_STT_2.Q AND NOT #"PLUS BIT"[32];   // rising edge
   #"PLUS BIT"[32] := #FILL_STT_2.Q;
   IF #_w2 AND #AUTO THEN #FILL_STT_SEQ2 := TRUE; END_IF;
   IF #_w1 AND "Tag_75" THEN #GUN_DOWN2 := TRUE; END_IF;
END_REGION

REGION Network 18: CYL 3 LOCK
   RUNG wire#powerrail
      Contact( "AlwaysTRUE" )
      Contact( #ENABLE_CYLINDER[3] )
      Contact( #CYCLE_OK )
      wire#w1
      Contact( #FIRST_CYCLE )
      { S7_Templates := "SrcType := Int" } EQ_Contact(in1 := #CYL_COUNTER_S3.CV, in2 := #First_Cylinder[3])
      wire#w2
      S_Coil( #"LIFT TABLE3" )
      { S7_Templates := "time_type := Time" } #FILL_STT_3.TON(pt := T#0S, et =>)
      P_Trig( #"PLUS BIT"[33] )
      Contact( #AUTO )
      S_Coil( #FILL_STT_SEQ3 )
   END_RUNG
   RUNG wire#w1
      Contact( #CYCLE_RESTART )
      { S7_Templates := "SrcType := Int" } EQ_Contact(in1 := #CYL_COUNT_CONT_S3.CV, in2 := #"CYL COUNT  VALUE")
   END_RUNG wire#w2
   RUNG wire#w2
      Contact( "Tag_75" )
      S_Coil( #GUN_DOWN3 )
   END_RUNG
   // the same network as SCL:
   #_w1 := "AlwaysTRUE" AND #ENABLE_CYLINDER[3] AND #CYCLE_OK AND ((#FIRST_CYCLE AND (#CYL_COUNTER_S3.CV = #First_Cylinder[3])) OR (#CYCLE_RESTART AND (#CYL_COUNT_CONT_S3.CV = #"CYL COUNT  VALUE")));
   IF #_w1 THEN #"LIFT TABLE3" := TRUE; END_IF;
   #FILL_STT_3(IN := #_w1, PT := T#0S);   // TON
   #_w2 := #FILL_STT_3.Q AND NOT #"PLUS BIT"[33];   // rising edge
   #"PLUS BIT"[33] := #FILL_STT_3.Q;
   IF #_w2 AND #AUTO THEN #FILL_STT_SEQ3 := TRUE; END_IF;
   IF #_w1 AND "Tag_75" THEN #GUN_DOWN3 := TRUE; END_IF;
END_REGION

REGION Network 19: CYL 4 LOCK
   RUNG wire#powerrail
      Contact( "AlwaysTRUE" )
      Contact( #ENABLE_CYLINDER[4] )
      Contact( #CYCLE_OK )
      wire#w1
      Contact( #FIRST_CYCLE )
      { S7_Templates := "SrcType := Int" } EQ_Contact(in1 := #CYL_COUNTER_S4.CV, in2 := #First_Cylinder[4])
      wire#w2
      S_Coil( #"LIFT TABLE4" )
      { S7_Templates := "time_type := Time" } #FILL_STT_4.TON(pt := T#0S, et =>)
      P_Trig( #"PLUS BIT"[34] )
      Contact( #AUTO )
      S_Coil( #FILL_STT_SEQ4 )
   END_RUNG
   RUNG wire#w1
      Contact( #CYCLE_RESTART )
      { S7_Templates := "SrcType := Int" } EQ_Contact(in1 := #CYL_COUNT_CONT_S4.CV, in2 := #"CYL COUNT  VALUE")
   END_RUNG wire#w2
   RUNG wire#w2
      Contact( "Tag_75" )
      S_Coil( #GUN_DOWN4 )
   END_RUNG
   // the same network as SCL:
   #_w1 := "AlwaysTRUE" AND #ENABLE_CYLINDER[4] AND #CYCLE_OK AND ((#FIRST_CYCLE AND (#CYL_COUNTER_S4.CV = #First_Cylinder[4])) OR (#CYCLE_RESTART AND (#CYL_COUNT_CONT_S4.CV = #"CYL COUNT  VALUE")));
   IF #_w1 THEN #"LIFT TABLE4" := TRUE; END_IF;
   #FILL_STT_4(IN := #_w1, PT := T#0S);   // TON
   #_w2 := #FILL_STT_4.Q AND NOT #"PLUS BIT"[34];   // rising edge
   #"PLUS BIT"[34] := #FILL_STT_4.Q;
   IF #_w2 AND #AUTO THEN #FILL_STT_SEQ4 := TRUE; END_IF;
   IF #_w1 AND "Tag_75" THEN #GUN_DOWN4 := TRUE; END_IF;
END_REGION

REGION Network 20: CYL 5 LOCK
   RUNG wire#powerrail
      Contact( "AlwaysTRUE" )
      Contact( #ENABLE_CYLINDER[5] )
      Contact( #CYCLE_OK )
      wire#w1
      Contact( #FIRST_CYCLE )
      { S7_Templates := "SrcType := Int" } EQ_Contact(in1 := #CYL_COUNTER_S5.CV, in2 := #First_Cylinder[5])
      wire#w2
      S_Coil( #"LIFT TABLE5" )
      { S7_Templates := "time_type := Time" } #FILL_STT_5.TON(pt := T#0S, et =>)
      P_Trig( #"PLUS BIT"[35] )
      Contact( #AUTO )
      S_Coil( #FILL_STT_SEQ5 )
   END_RUNG
   RUNG wire#w1
      Contact( #CYCLE_RESTART )
      { S7_Templates := "SrcType := Int" } EQ_Contact(in1 := #CYL_COUNT_CONT_S5.CV, in2 := #"CYL COUNT  VALUE")
   END_RUNG wire#w2
   RUNG wire#w2
      Contact( "Tag_75" )
      S_Coil( #GUN_DOWN5 )
   END_RUNG
   // the same network as SCL:
   #_w1 := "AlwaysTRUE" AND #ENABLE_CYLINDER[5] AND #CYCLE_OK AND ((#FIRST_CYCLE AND (#CYL_COUNTER_S5.CV = #First_Cylinder[5])) OR (#CYCLE_RESTART AND (#CYL_COUNT_CONT_S5.CV = #"CYL COUNT  VALUE")));
   IF #_w1 THEN #"LIFT TABLE5" := TRUE; END_IF;
   #FILL_STT_5(IN := #_w1, PT := T#0S);   // TON
   #_w2 := #FILL_STT_5.Q AND NOT #"PLUS BIT"[35];   // rising edge
   #"PLUS BIT"[35] := #FILL_STT_5.Q;
   IF #_w2 AND #AUTO THEN #FILL_STT_SEQ5 := TRUE; END_IF;
   IF #_w1 AND "Tag_75" THEN #GUN_DOWN5 := TRUE; END_IF;
END_REGION

REGION Network 21: CYL 6 LOCK
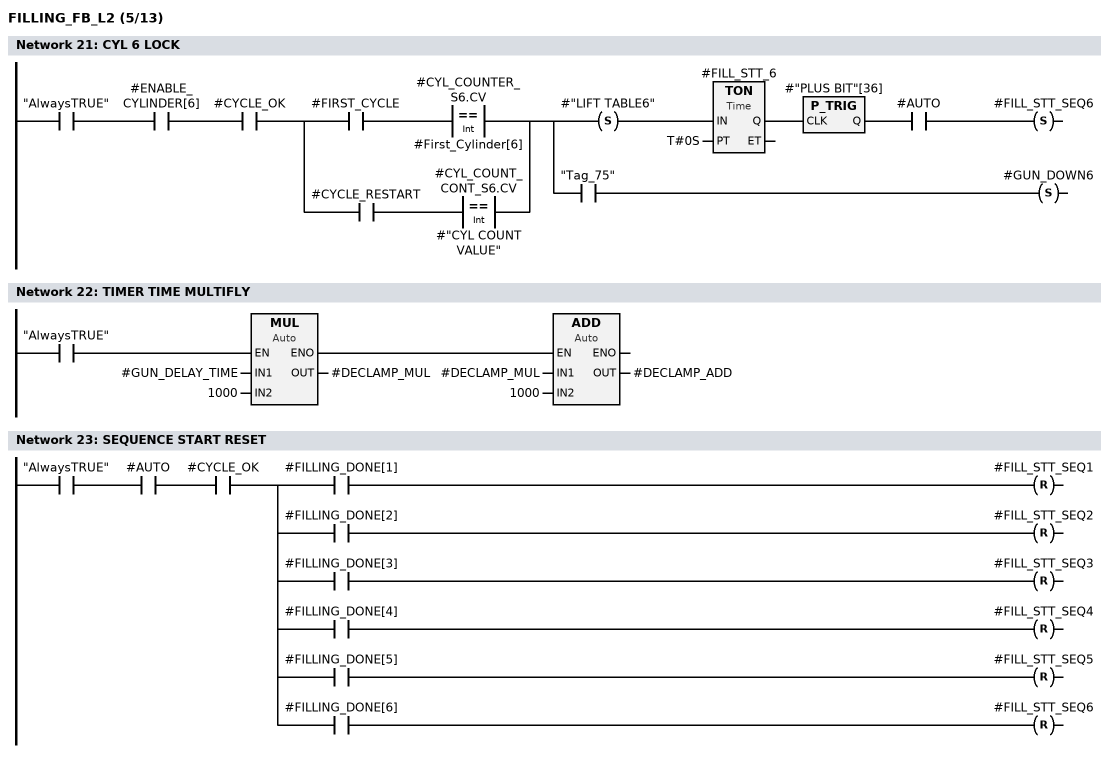
   RUNG wire#powerrail
      Contact( "AlwaysTRUE" )
      Contact( #ENABLE_CYLINDER[6] )
      Contact( #CYCLE_OK )
      wire#w1
      Contact( #FIRST_CYCLE )
      { S7_Templates := "SrcType := Int" } EQ_Contact(in1 := #CYL_COUNTER_S6.CV, in2 := #First_Cylinder[6])
      wire#w2
      S_Coil( #"LIFT TABLE6" )
      { S7_Templates := "time_type := Time" } #FILL_STT_6.TON(pt := T#0S, et =>)
      P_Trig( #"PLUS BIT"[36] )
      Contact( #AUTO )
      S_Coil( #FILL_STT_SEQ6 )
   END_RUNG
   RUNG wire#w1
      Contact( #CYCLE_RESTART )
      { S7_Templates := "SrcType := Int" } EQ_Contact(in1 := #CYL_COUNT_CONT_S6.CV, in2 := #"CYL COUNT  VALUE")
   END_RUNG wire#w2
   RUNG wire#w2
      Contact( "Tag_75" )
      S_Coil( #GUN_DOWN6 )
   END_RUNG
   // the same network as SCL:
   #_w1 := "AlwaysTRUE" AND #ENABLE_CYLINDER[6] AND #CYCLE_OK AND ((#FIRST_CYCLE AND (#CYL_COUNTER_S6.CV = #First_Cylinder[6])) OR (#CYCLE_RESTART AND (#CYL_COUNT_CONT_S6.CV = #"CYL COUNT  VALUE")));
   IF #_w1 THEN #"LIFT TABLE6" := TRUE; END_IF;
   #FILL_STT_6(IN := #_w1, PT := T#0S);   // TON
   #_w2 := #FILL_STT_6.Q AND NOT #"PLUS BIT"[36];   // rising edge
   #"PLUS BIT"[36] := #FILL_STT_6.Q;
   IF #_w2 AND #AUTO THEN #FILL_STT_SEQ6 := TRUE; END_IF;
   IF #_w1 AND "Tag_75" THEN #GUN_DOWN6 := TRUE; END_IF;
END_REGION

REGION Network 22: TIMER TIME MULTIFLY
   RUNG wire#powerrail
      Contact( "AlwaysTRUE" )
      Mul(in1 := #GUN_DELAY_TIME, in2 := 1000, out => #DECLAMP_MUL)
      Add(in1 := #DECLAMP_MUL, in2 := 1000, out => #DECLAMP_ADD)
   END_RUNG
   // the same network as SCL:
   IF "AlwaysTRUE" THEN
       #DECLAMP_MUL := #GUN_DELAY_TIME * 1000;
       #DECLAMP_ADD := #DECLAMP_MUL + 1000;
   END_IF;
END_REGION

REGION Network 23: SEQUENCE START RESET
   RUNG wire#powerrail
      Contact( "AlwaysTRUE" )
      Contact( #AUTO )
      Contact( #CYCLE_OK )
      wire#w1
      Contact( #FILLING_DONE[1] )
      R_Coil( #FILL_STT_SEQ1 )
   END_RUNG
   RUNG wire#w1
      Contact( #FILLING_DONE[2] )
      R_Coil( #FILL_STT_SEQ2 )
   END_RUNG
   RUNG wire#w1
      Contact( #FILLING_DONE[3] )
      R_Coil( #FILL_STT_SEQ3 )
   END_RUNG
   RUNG wire#w1
      Contact( #FILLING_DONE[4] )
      R_Coil( #FILL_STT_SEQ4 )
   END_RUNG
   RUNG wire#w1
      Contact( #FILLING_DONE[5] )
      R_Coil( #FILL_STT_SEQ5 )
   END_RUNG
   RUNG wire#w1
      Contact( #FILLING_DONE[6] )
      R_Coil( #FILL_STT_SEQ6 )
   END_RUNG
   // the same network as SCL:
   #_w1 := "AlwaysTRUE" AND #AUTO AND #CYCLE_OK;
   IF #_w1 AND #FILLING_DONE[1] THEN #FILL_STT_SEQ1 := FALSE; END_IF;
   IF #_w1 AND #FILLING_DONE[2] THEN #FILL_STT_SEQ2 := FALSE; END_IF;
   IF #_w1 AND #FILLING_DONE[3] THEN #FILL_STT_SEQ3 := FALSE; END_IF;
   IF #_w1 AND #FILLING_DONE[4] THEN #FILL_STT_SEQ4 := FALSE; END_IF;
   IF #_w1 AND #FILLING_DONE[5] THEN #FILL_STT_SEQ5 := FALSE; END_IF;
   IF #_w1 AND #FILLING_DONE[6] THEN #FILL_STT_SEQ6 := FALSE; END_IF;
END_REGION

REGION Network 24: GUN RESET
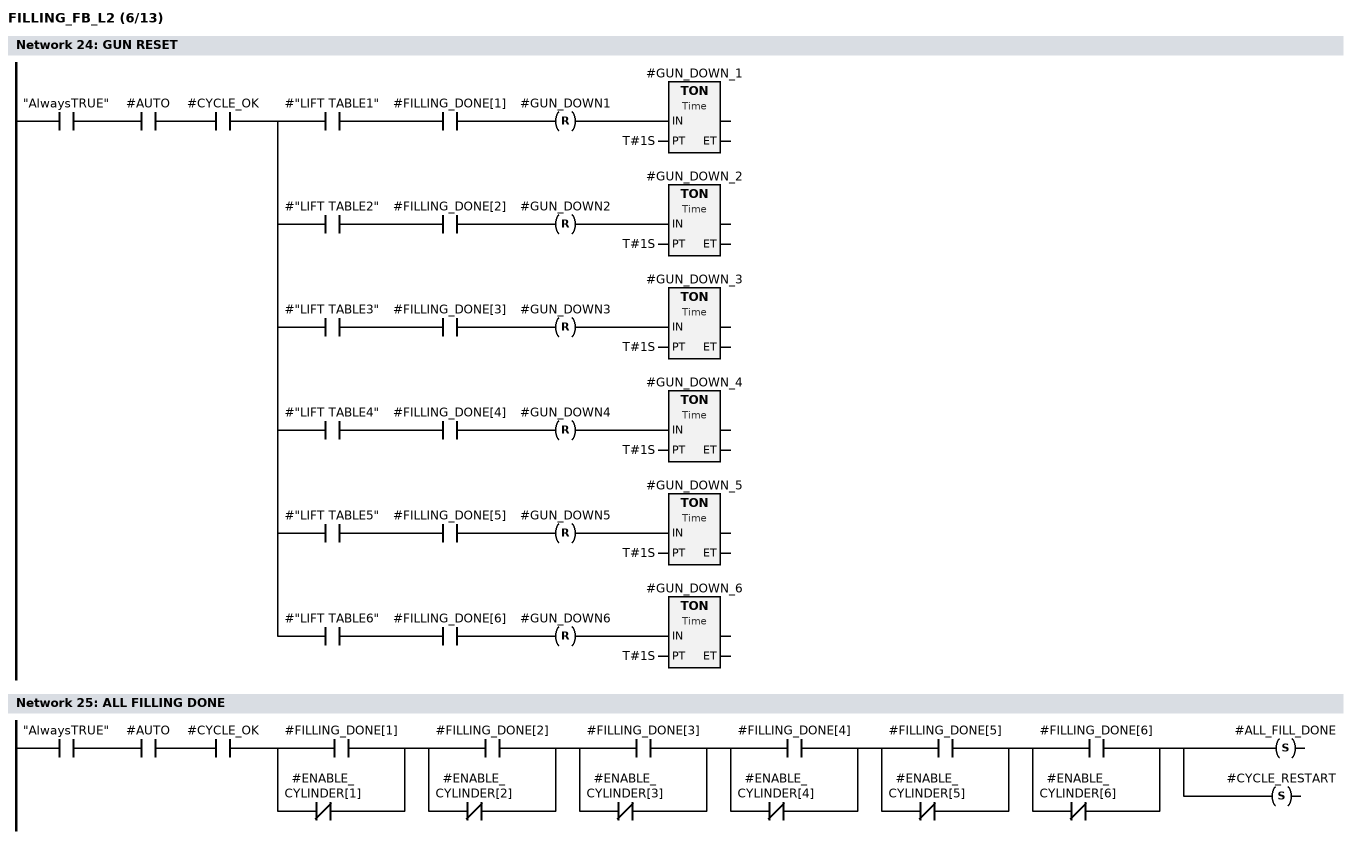
   RUNG wire#powerrail
      Contact( "AlwaysTRUE" )
      Contact( #AUTO )
      Contact( #CYCLE_OK )
      wire#w1
      Contact( #"LIFT TABLE1" )
      Contact( #FILLING_DONE[1] )
      R_Coil( #GUN_DOWN1 )
      { S7_Templates := "time_type := Time" } #GUN_DOWN_1.TON(pt := T#1S, et =>)
   END_RUNG
   RUNG wire#w1
      Contact( #"LIFT TABLE2" )
      Contact( #FILLING_DONE[2] )
      R_Coil( #GUN_DOWN2 )
      { S7_Templates := "time_type := Time" } #GUN_DOWN_2.TON(pt := T#1S, et =>)
   END_RUNG
   RUNG wire#w1
      Contact( #"LIFT TABLE3" )
      Contact( #FILLING_DONE[3] )
      R_Coil( #GUN_DOWN3 )
      { S7_Templates := "time_type := Time" } #GUN_DOWN_3.TON(pt := T#1S, et =>)
   END_RUNG
   RUNG wire#w1
      Contact( #"LIFT TABLE4" )
      Contact( #FILLING_DONE[4] )
      R_Coil( #GUN_DOWN4 )
      { S7_Templates := "time_type := Time" } #GUN_DOWN_4.TON(pt := T#1S, et =>)
   END_RUNG
   RUNG wire#w1
      Contact( #"LIFT TABLE5" )
      Contact( #FILLING_DONE[5] )
      R_Coil( #GUN_DOWN5 )
      { S7_Templates := "time_type := Time" } #GUN_DOWN_5.TON(pt := T#1S, et =>)
   END_RUNG
   RUNG wire#w1
      Contact( #"LIFT TABLE6" )
      Contact( #FILLING_DONE[6] )
      R_Coil( #GUN_DOWN6 )
      { S7_Templates := "time_type := Time" } #GUN_DOWN_6.TON(pt := T#1S, et =>)
   END_RUNG
   // the same network as SCL:
   #_w1 := "AlwaysTRUE" AND #AUTO AND #CYCLE_OK;
   #_w2 := #_w1 AND #"LIFT TABLE1" AND #FILLING_DONE[1];
   IF #_w2 THEN #GUN_DOWN1 := FALSE; END_IF;
   #GUN_DOWN_1(IN := #_w2, PT := T#1S);   // TON
   #_w3 := #_w1 AND #"LIFT TABLE2" AND #FILLING_DONE[2];
   IF #_w3 THEN #GUN_DOWN2 := FALSE; END_IF;
   #GUN_DOWN_2(IN := #_w3, PT := T#1S);   // TON
   #_w4 := #_w1 AND #"LIFT TABLE3" AND #FILLING_DONE[3];
   IF #_w4 THEN #GUN_DOWN3 := FALSE; END_IF;
   #GUN_DOWN_3(IN := #_w4, PT := T#1S);   // TON
   #_w5 := #_w1 AND #"LIFT TABLE4" AND #FILLING_DONE[4];
   IF #_w5 THEN #GUN_DOWN4 := FALSE; END_IF;
   #GUN_DOWN_4(IN := #_w5, PT := T#1S);   // TON
   #_w6 := #_w1 AND #"LIFT TABLE5" AND #FILLING_DONE[5];
   IF #_w6 THEN #GUN_DOWN5 := FALSE; END_IF;
   #GUN_DOWN_5(IN := #_w6, PT := T#1S);   // TON
   #_w7 := #_w1 AND #"LIFT TABLE6" AND #FILLING_DONE[6];
   IF #_w7 THEN #GUN_DOWN6 := FALSE; END_IF;
   #GUN_DOWN_6(IN := #_w7, PT := T#1S);   // TON
END_REGION

REGION Network 25: ALL FILLING DONE
   RUNG wire#powerrail
      Contact( "AlwaysTRUE" )
      Contact( #AUTO )
      Contact( #CYCLE_OK )
      wire#w1
      Contact( #FILLING_DONE[1] )
      wire#w2
      Contact( #FILLING_DONE[2] )
      wire#w3
      Contact( #FILLING_DONE[3] )
      wire#w4
      Contact( #FILLING_DONE[4] )
      wire#w5
      Contact( #FILLING_DONE[5] )
      wire#w6
      Contact( #FILLING_DONE[6] )
      wire#w7
      S_Coil( #ALL_FILL_DONE )
   END_RUNG
   RUNG wire#w1
      I_Contact( #ENABLE_CYLINDER[1] )
   END_RUNG wire#w2
   RUNG wire#w2
      I_Contact( #ENABLE_CYLINDER[2] )
   END_RUNG wire#w3
   RUNG wire#w3
      I_Contact( #ENABLE_CYLINDER[3] )
   END_RUNG wire#w4
   RUNG wire#w4
      I_Contact( #ENABLE_CYLINDER[4] )
   END_RUNG wire#w5
   RUNG wire#w5
      I_Contact( #ENABLE_CYLINDER[5] )
   END_RUNG wire#w6
   RUNG wire#w6
      I_Contact( #ENABLE_CYLINDER[6] )
   END_RUNG wire#w7
   RUNG wire#w7
      S_Coil( #CYCLE_RESTART )
   END_RUNG
   // the same network as SCL:
   IF "AlwaysTRUE" AND #AUTO AND #CYCLE_OK AND (#FILLING_DONE[1] OR NOT #ENABLE_CYLINDER[1]) AND (#FILLING_DONE[2] OR NOT #ENABLE_CYLINDER[2]) AND (#FILLING_DONE[3] OR NOT #ENABLE_CYLINDER[3]) AND (#FILLING_DONE[4] OR NOT #ENABLE_CYLINDER[4]) AND (#FILLING_DONE[5] OR NOT #ENABLE_CYLINDER[5]) AND (#FILLING_DONE[6] OR NOT #ENABLE_CYLINDER[6]) THEN
       #ALL_FILL_DONE := TRUE;
       #CYCLE_RESTART := TRUE;
   END_IF;
END_REGION

REGION Network 26: ALL GUN UP
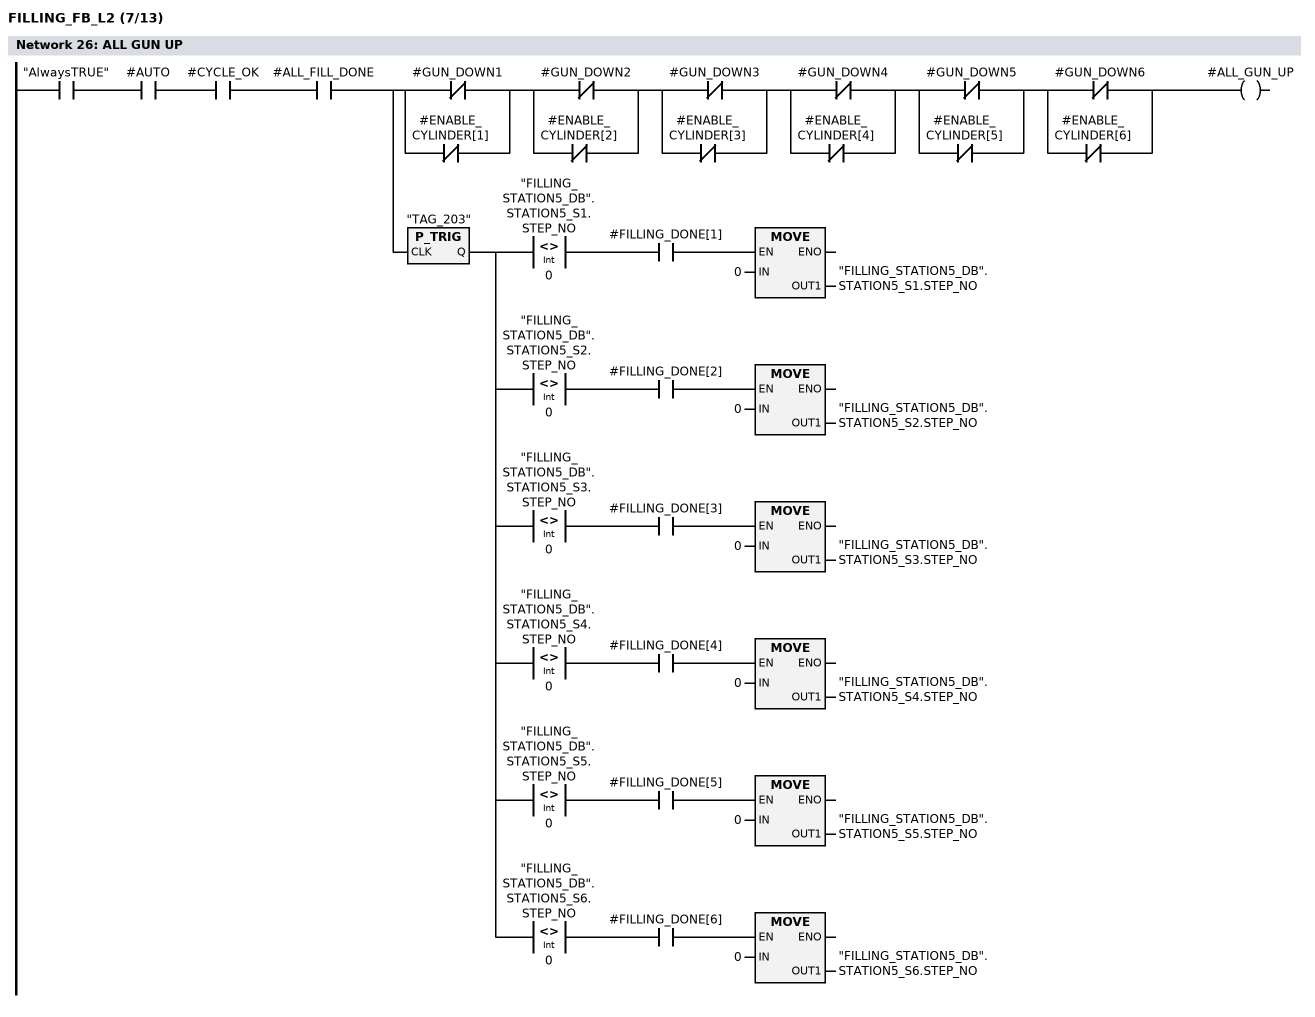
   RUNG wire#powerrail
      Contact( "AlwaysTRUE" )
      Contact( #AUTO )
      Contact( #CYCLE_OK )
      Contact( #ALL_FILL_DONE )
      wire#w1
      I_Contact( #GUN_DOWN1 )
      wire#w2
      I_Contact( #GUN_DOWN2 )
      wire#w3
      I_Contact( #GUN_DOWN3 )
      wire#w4
      I_Contact( #GUN_DOWN4 )
      wire#w5
      I_Contact( #GUN_DOWN5 )
      wire#w6
      I_Contact( #GUN_DOWN6 )
      wire#w7
      Coil( #ALL_GUN_UP )
   END_RUNG
   RUNG wire#w1
      I_Contact( #ENABLE_CYLINDER[1] )
   END_RUNG wire#w2
   RUNG wire#w2
      I_Contact( #ENABLE_CYLINDER[2] )
   END_RUNG wire#w3
   RUNG wire#w3
      I_Contact( #ENABLE_CYLINDER[3] )
   END_RUNG wire#w4
   RUNG wire#w4
      I_Contact( #ENABLE_CYLINDER[4] )
   END_RUNG wire#w5
   RUNG wire#w5
      I_Contact( #ENABLE_CYLINDER[5] )
   END_RUNG wire#w6
   RUNG wire#w6
      I_Contact( #ENABLE_CYLINDER[6] )
   END_RUNG wire#w7
   RUNG wire#w1
      P_Trig( "TAG_203" )
      wire#w8
      { S7_Templates := "SrcType := Int" } NE_Contact(in1 := "FILLING_STATION5_DB".STATION5_S1.STEP_NO, in2 := 0)
      Contact( #FILLING_DONE[1] )
      Move(in := 0, out1 => "FILLING_STATION5_DB".STATION5_S1.STEP_NO)
   END_RUNG
   RUNG wire#w8
      { S7_Templates := "SrcType := Int" } NE_Contact(in1 := "FILLING_STATION5_DB".STATION5_S2.STEP_NO, in2 := 0)
      Contact( #FILLING_DONE[2] )
      Move(in := 0, out1 => "FILLING_STATION5_DB".STATION5_S2.STEP_NO)
   END_RUNG
   RUNG wire#w8
      { S7_Templates := "SrcType := Int" } NE_Contact(in1 := "FILLING_STATION5_DB".STATION5_S3.STEP_NO, in2 := 0)
      Contact( #FILLING_DONE[3] )
      Move(in := 0, out1 => "FILLING_STATION5_DB".STATION5_S3.STEP_NO)
   END_RUNG
   RUNG wire#w8
      { S7_Templates := "SrcType := Int" } NE_Contact(in1 := "FILLING_STATION5_DB".STATION5_S4.STEP_NO, in2 := 0)
      Contact( #FILLING_DONE[4] )
      Move(in := 0, out1 => "FILLING_STATION5_DB".STATION5_S4.STEP_NO)
   END_RUNG
   RUNG wire#w8
      { S7_Templates := "SrcType := Int" } NE_Contact(in1 := "FILLING_STATION5_DB".STATION5_S5.STEP_NO, in2 := 0)
      Contact( #FILLING_DONE[5] )
      Move(in := 0, out1 => "FILLING_STATION5_DB".STATION5_S5.STEP_NO)
   END_RUNG
   RUNG wire#w8
      { S7_Templates := "SrcType := Int" } NE_Contact(in1 := "FILLING_STATION5_DB".STATION5_S6.STEP_NO, in2 := 0)
      Contact( #FILLING_DONE[6] )
      Move(in := 0, out1 => "FILLING_STATION5_DB".STATION5_S6.STEP_NO)
   END_RUNG
   // the same network as SCL:
   #_w1 := "AlwaysTRUE" AND #AUTO AND #CYCLE_OK AND #ALL_FILL_DONE;
   #ALL_GUN_UP := #_w1 AND (NOT #GUN_DOWN1 OR NOT #ENABLE_CYLINDER[1]) AND (NOT #GUN_DOWN2 OR NOT #ENABLE_CYLINDER[2]) AND (NOT #GUN_DOWN3 OR NOT #ENABLE_CYLINDER[3]) AND (NOT #GUN_DOWN4 OR NOT #ENABLE_CYLINDER[4]) AND (NOT #GUN_DOWN5 OR NOT #ENABLE_CYLINDER[5]) AND (NOT #GUN_DOWN6 OR NOT #ENABLE_CYLINDER[6]);
   #_w2 := #_w1 AND NOT "TAG_203";   // rising edge
   "TAG_203" := #_w1;
   IF #_w2 AND ("FILLING_STATION5_DB".STATION5_S1.STEP_NO <> 0) AND #FILLING_DONE[1] THEN
       "FILLING_STATION5_DB".STATION5_S1.STEP_NO := 0;
   END_IF;
   IF #_w2 AND ("FILLING_STATION5_DB".STATION5_S2.STEP_NO <> 0) AND #FILLING_DONE[2] THEN
       "FILLING_STATION5_DB".STATION5_S2.STEP_NO := 0;
   END_IF;
   IF #_w2 AND ("FILLING_STATION5_DB".STATION5_S3.STEP_NO <> 0) AND #FILLING_DONE[3] THEN
       "FILLING_STATION5_DB".STATION5_S3.STEP_NO := 0;
   END_IF;
   IF #_w2 AND ("FILLING_STATION5_DB".STATION5_S4.STEP_NO <> 0) AND #FILLING_DONE[4] THEN
       "FILLING_STATION5_DB".STATION5_S4.STEP_NO := 0;
   END_IF;
   IF #_w2 AND ("FILLING_STATION5_DB".STATION5_S5.STEP_NO <> 0) AND #FILLING_DONE[5] THEN
       "FILLING_STATION5_DB".STATION5_S5.STEP_NO := 0;
   END_IF;
   IF #_w2 AND ("FILLING_STATION5_DB".STATION5_S6.STEP_NO <> 0) AND #FILLING_DONE[6] THEN
       "FILLING_STATION5_DB".STATION5_S6.STEP_NO := 0;
   END_IF;
END_REGION

REGION Network 27: CYCLE COMPLETED
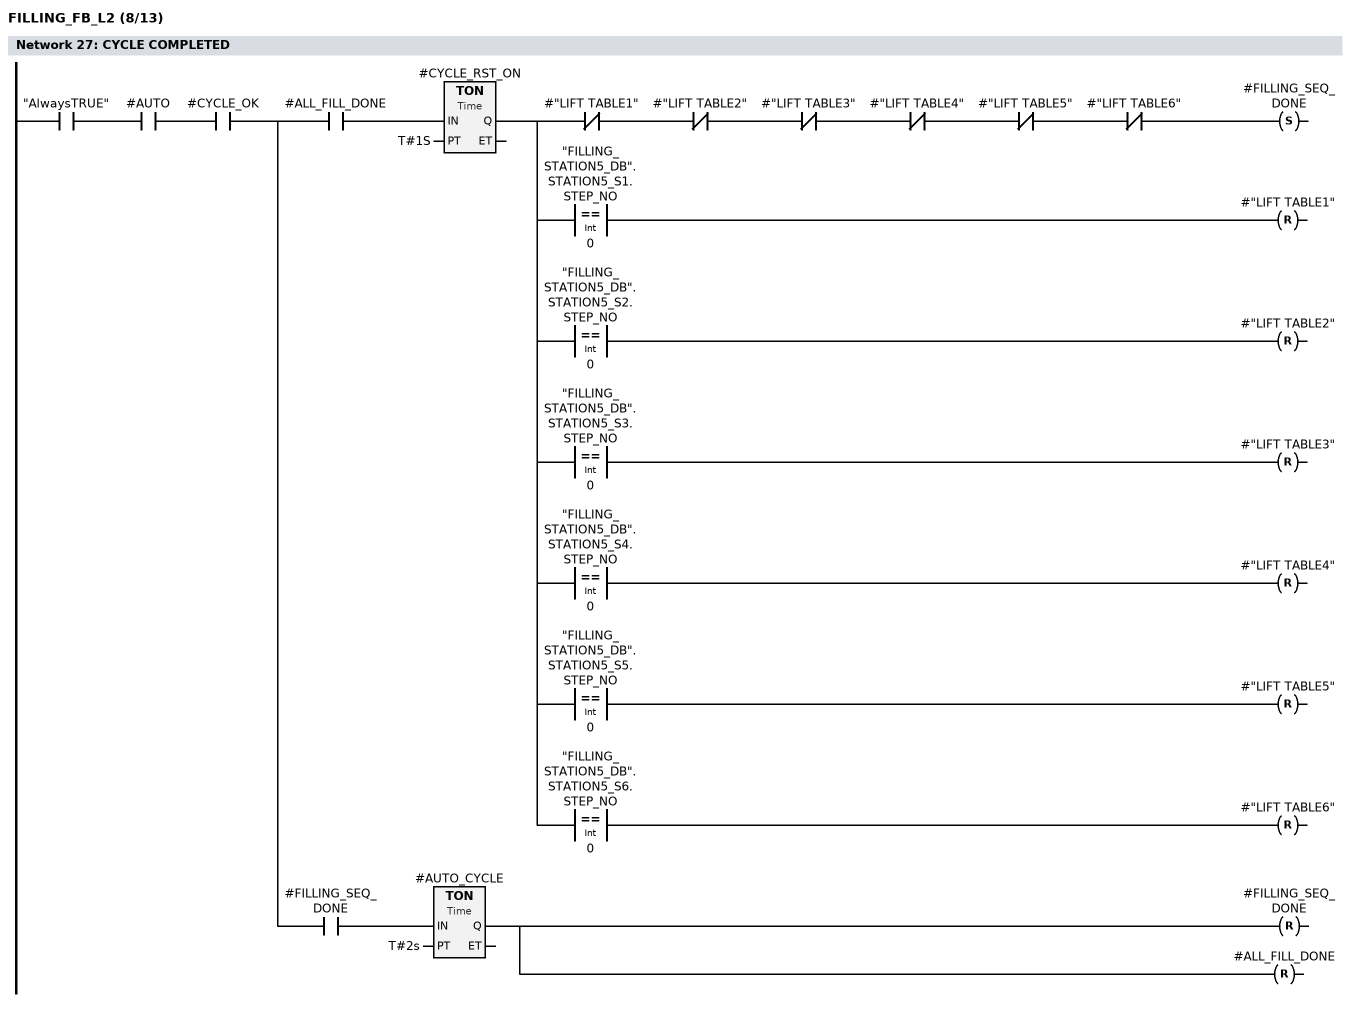
   RUNG wire#powerrail
      Contact( "AlwaysTRUE" )
      Contact( #AUTO )
      Contact( #CYCLE_OK )
      wire#w1
      Contact( #ALL_FILL_DONE )
      { S7_Templates := "time_type := Time" } #CYCLE_RST_ON.TON(pt := T#1S, et =>)
      wire#w2
      I_Contact( #"LIFT TABLE1" )
      I_Contact( #"LIFT TABLE2" )
      I_Contact( #"LIFT TABLE3" )
      I_Contact( #"LIFT TABLE4" )
      I_Contact( #"LIFT TABLE5" )
      I_Contact( #"LIFT TABLE6" )
      S_Coil( #FILLING_SEQ_DONE )
   END_RUNG
   RUNG wire#w2
      { S7_Templates := "SrcType := Int" } EQ_Contact(in1 := "FILLING_STATION5_DB".STATION5_S1.STEP_NO, in2 := 0)
      R_Coil( #"LIFT TABLE1" )
   END_RUNG
   RUNG wire#w2
      { S7_Templates := "SrcType := Int" } EQ_Contact(in1 := "FILLING_STATION5_DB".STATION5_S2.STEP_NO, in2 := 0)
      R_Coil( #"LIFT TABLE2" )
   END_RUNG
   RUNG wire#w2
      { S7_Templates := "SrcType := Int" } EQ_Contact(in1 := "FILLING_STATION5_DB".STATION5_S3.STEP_NO, in2 := 0)
      R_Coil( #"LIFT TABLE3" )
   END_RUNG
   RUNG wire#w2
      { S7_Templates := "SrcType := Int" } EQ_Contact(in1 := "FILLING_STATION5_DB".STATION5_S4.STEP_NO, in2 := 0)
      R_Coil( #"LIFT TABLE4" )
   END_RUNG
   RUNG wire#w2
      { S7_Templates := "SrcType := Int" } EQ_Contact(in1 := "FILLING_STATION5_DB".STATION5_S5.STEP_NO, in2 := 0)
      R_Coil( #"LIFT TABLE5" )
   END_RUNG
   RUNG wire#w2
      { S7_Templates := "SrcType := Int" } EQ_Contact(in1 := "FILLING_STATION5_DB".STATION5_S6.STEP_NO, in2 := 0)
      R_Coil( #"LIFT TABLE6" )
   END_RUNG
   RUNG wire#w1
      Contact( #FILLING_SEQ_DONE )
      { S7_Templates := "time_type := Time" } #AUTO_CYCLE.TON(pt := T#2s, et =>)
      wire#w3
      R_Coil( #FILLING_SEQ_DONE )
   END_RUNG
   RUNG wire#w3
      R_Coil( #ALL_FILL_DONE )
   END_RUNG
   // the same network as SCL:
   #_w1 := "AlwaysTRUE" AND #AUTO AND #CYCLE_OK;
   #CYCLE_RST_ON(IN := #_w1 AND #ALL_FILL_DONE, PT := T#1S);   // TON
   IF #CYCLE_RST_ON.Q AND NOT #"LIFT TABLE1" AND NOT #"LIFT TABLE2" AND NOT #"LIFT TABLE3" AND NOT #"LIFT TABLE4" AND NOT #"LIFT TABLE5" AND NOT #"LIFT TABLE6" THEN
       #FILLING_SEQ_DONE := TRUE;
   END_IF;
   IF #CYCLE_RST_ON.Q AND ("FILLING_STATION5_DB".STATION5_S1.STEP_NO = 0) THEN
       #"LIFT TABLE1" := FALSE;
   END_IF;
   IF #CYCLE_RST_ON.Q AND ("FILLING_STATION5_DB".STATION5_S2.STEP_NO = 0) THEN
       #"LIFT TABLE2" := FALSE;
   END_IF;
   IF #CYCLE_RST_ON.Q AND ("FILLING_STATION5_DB".STATION5_S3.STEP_NO = 0) THEN
       #"LIFT TABLE3" := FALSE;
   END_IF;
   IF #CYCLE_RST_ON.Q AND ("FILLING_STATION5_DB".STATION5_S4.STEP_NO = 0) THEN
       #"LIFT TABLE4" := FALSE;
   END_IF;
   IF #CYCLE_RST_ON.Q AND ("FILLING_STATION5_DB".STATION5_S5.STEP_NO = 0) THEN
       #"LIFT TABLE5" := FALSE;
   END_IF;
   IF #CYCLE_RST_ON.Q AND ("FILLING_STATION5_DB".STATION5_S6.STEP_NO = 0) THEN
       #"LIFT TABLE6" := FALSE;
   END_IF;
   #AUTO_CYCLE(IN := #_w1 AND #FILLING_SEQ_DONE, PT := T#2s);   // TON
   IF #AUTO_CYCLE.Q THEN
       #FILLING_SEQ_DONE := FALSE;
       #ALL_FILL_DONE := FALSE;
   END_IF;
END_REGION

REGION Network 28: CYCLE RESET
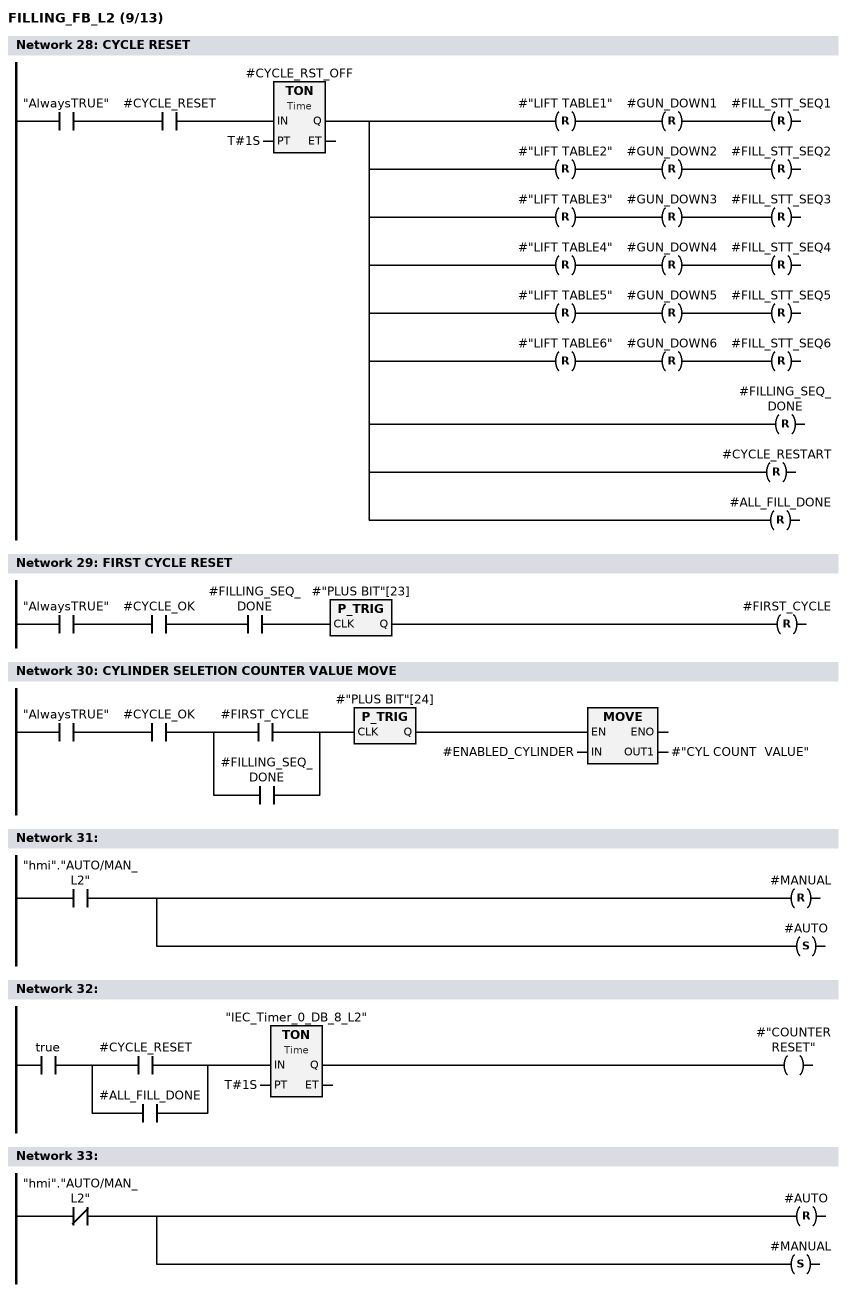
   RUNG wire#powerrail
      Contact( "AlwaysTRUE" )
      Contact( #CYCLE_RESET )
      { S7_Templates := "time_type := Time" } #CYCLE_RST_OFF.TON(pt := T#1S, et =>)
      wire#w1
      R_Coil( #"LIFT TABLE1" )
      R_Coil( #GUN_DOWN1 )
      R_Coil( #FILL_STT_SEQ1 )
   END_RUNG
   RUNG wire#w1
      R_Coil( #"LIFT TABLE2" )
      R_Coil( #GUN_DOWN2 )
      R_Coil( #FILL_STT_SEQ2 )
   END_RUNG
   RUNG wire#w1
      R_Coil( #"LIFT TABLE3" )
      R_Coil( #GUN_DOWN3 )
      R_Coil( #FILL_STT_SEQ3 )
   END_RUNG
   RUNG wire#w1
      R_Coil( #"LIFT TABLE4" )
      R_Coil( #GUN_DOWN4 )
      R_Coil( #FILL_STT_SEQ4 )
   END_RUNG
   RUNG wire#w1
      R_Coil( #"LIFT TABLE5" )
      R_Coil( #GUN_DOWN5 )
      R_Coil( #FILL_STT_SEQ5 )
   END_RUNG
   RUNG wire#w1
      R_Coil( #"LIFT TABLE6" )
      R_Coil( #GUN_DOWN6 )
      R_Coil( #FILL_STT_SEQ6 )
   END_RUNG
   RUNG wire#w1
      R_Coil( #FILLING_SEQ_DONE )
   END_RUNG
   RUNG wire#w1
      R_Coil( #CYCLE_RESTART )
   END_RUNG
   RUNG wire#w1
      R_Coil( #ALL_FILL_DONE )
   END_RUNG
   // the same network as SCL:
   #CYCLE_RST_OFF(IN := "AlwaysTRUE" AND #CYCLE_RESET, PT := T#1S);   // TON
   IF #CYCLE_RST_OFF.Q THEN
       #"LIFT TABLE1" := FALSE;
       #GUN_DOWN1 := FALSE;
       #FILL_STT_SEQ1 := FALSE;
       #"LIFT TABLE2" := FALSE;
       #GUN_DOWN2 := FALSE;
       #FILL_STT_SEQ2 := FALSE;
       #"LIFT TABLE3" := FALSE;
       #GUN_DOWN3 := FALSE;
       #FILL_STT_SEQ3 := FALSE;
       #"LIFT TABLE4" := FALSE;
       #GUN_DOWN4 := FALSE;
       #FILL_STT_SEQ4 := FALSE;
       #"LIFT TABLE5" := FALSE;
       #GUN_DOWN5 := FALSE;
       #FILL_STT_SEQ5 := FALSE;
       #"LIFT TABLE6" := FALSE;
       #GUN_DOWN6 := FALSE;
       #FILL_STT_SEQ6 := FALSE;
       #FILLING_SEQ_DONE := FALSE;
       #CYCLE_RESTART := FALSE;
       #ALL_FILL_DONE := FALSE;
   END_IF;
END_REGION

REGION Network 29: FIRST CYCLE RESET
   RUNG wire#powerrail
      Contact( "AlwaysTRUE" )
      Contact( #CYCLE_OK )
      Contact( #FILLING_SEQ_DONE )
      P_Trig( #"PLUS BIT"[23] )
      R_Coil( #FIRST_CYCLE )
   END_RUNG
   // the same network as SCL:
   #_w1 := "AlwaysTRUE" AND #CYCLE_OK AND #FILLING_SEQ_DONE;
   #_w2 := #_w1 AND NOT #"PLUS BIT"[23];   // rising edge
   #"PLUS BIT"[23] := #_w1;
   IF #_w2 THEN #FIRST_CYCLE := FALSE; END_IF;
END_REGION

REGION Network 30: CYLINDER SELETION COUNTER VALUE MOVE
   RUNG wire#powerrail
      Contact( "AlwaysTRUE" )
      Contact( #CYCLE_OK )
      wire#w1
      Contact( #FIRST_CYCLE )
      wire#w2
      P_Trig( #"PLUS BIT"[24] )
      Move(in := #ENABLED_CYLINDER, out1 => #"CYL COUNT  VALUE")
   END_RUNG
   RUNG wire#w1
      Contact( #FILLING_SEQ_DONE )
   END_RUNG wire#w2
   // the same network as SCL:
   #_w1 := "AlwaysTRUE" AND #CYCLE_OK AND (#FIRST_CYCLE OR #FILLING_SEQ_DONE);
   #_w2 := #_w1 AND NOT #"PLUS BIT"[24];   // rising edge
   #"PLUS BIT"[24] := #_w1;
   IF #_w2 THEN #"CYL COUNT  VALUE" := #ENABLED_CYLINDER; END_IF;
END_REGION

REGION Network 31
   RUNG wire#powerrail
      Contact( "hmi"."AUTO/MAN_L2" )
      wire#w1
      R_Coil( #MANUAL )
   END_RUNG
   RUNG wire#w1
      S_Coil( #AUTO )
   END_RUNG
   // the same network as SCL:
   IF "hmi"."AUTO/MAN_L2" THEN
       #MANUAL := FALSE;
       #AUTO := TRUE;
   END_IF;
END_REGION

REGION Network 32
   RUNG wire#powerrail
      Contact( true )
      wire#w1
      Contact( #CYCLE_RESET )
      wire#w2
      { S7_Templates := "time_type := Time" } "IEC_Timer_0_DB_8_L2".TON(pt := T#1S, et =>)
      Coil( #"COUNTER RESET" )
   END_RUNG
   RUNG wire#w1
      Contact( #ALL_FILL_DONE )
   END_RUNG wire#w2
   // the same network as SCL:
   "IEC_Timer_0_DB_8_L2".TON(IN := true AND (#CYCLE_RESET OR #ALL_FILL_DONE), PT := T#1S);
   #"COUNTER RESET" := "IEC_Timer_0_DB_8_L2".Q;
END_REGION

REGION Network 33
   RUNG wire#powerrail
      I_Contact( "hmi"."AUTO/MAN_L2" )
      wire#w1
      R_Coil( #AUTO )
   END_RUNG
   RUNG wire#w1
      S_Coil( #MANUAL )
   END_RUNG
   // the same network as SCL:
   IF NOT "hmi"."AUTO/MAN_L2" THEN
       #AUTO := FALSE;
       #MANUAL := TRUE;
   END_IF;
END_REGION

REGION Network 34
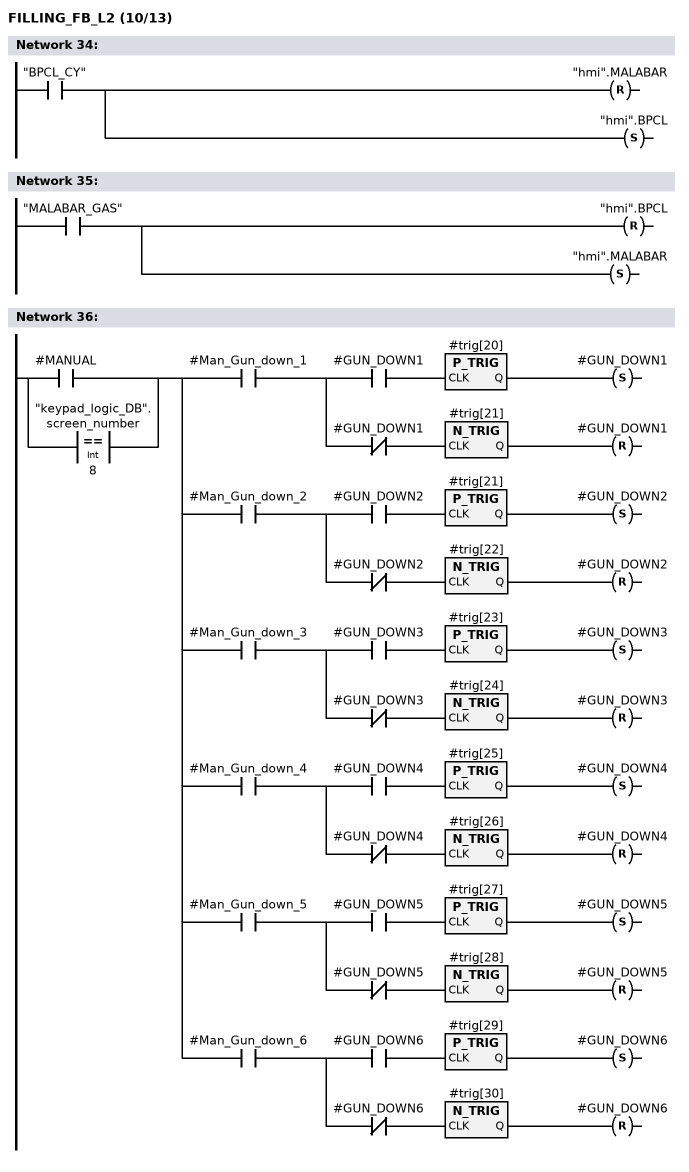
   RUNG wire#powerrail
      Contact( "BPCL_CY" )
      wire#w1
      R_Coil( "hmi".MALABAR )
   END_RUNG
   RUNG wire#w1
      S_Coil( "hmi".BPCL )
   END_RUNG
   // the same network as SCL:
   IF "BPCL_CY" THEN
       "hmi".MALABAR := FALSE;
       "hmi".BPCL := TRUE;
   END_IF;
END_REGION

REGION Network 35
   RUNG wire#powerrail
      Contact( "MALABAR_GAS" )
      wire#w1
      R_Coil( "hmi".BPCL )
   END_RUNG
   RUNG wire#w1
      S_Coil( "hmi".MALABAR )
   END_RUNG
   // the same network as SCL:
   IF "MALABAR_GAS" THEN
       "hmi".BPCL := FALSE;
       "hmi".MALABAR := TRUE;
   END_IF;
END_REGION

REGION Network 36
   RUNG wire#powerrail
      Contact( #MANUAL )
      wire#w1
      Contact( #Man_Gun_down_1 )
      wire#w2
      Contact( #GUN_DOWN1 )
      P_Trig( #trig[20] )
      S_Coil( #GUN_DOWN1 )
   END_RUNG
   RUNG wire#powerrail
      { S7_Templates := "SrcType := Int" } EQ_Contact(in1 := "keypad_logic_DB".screen_number, in2 := 8)
   END_RUNG wire#w1
   RUNG wire#w2
      I_Contact( #GUN_DOWN1 )
      N_Trig( #trig[21] )
      R_Coil( #GUN_DOWN1 )
   END_RUNG
   RUNG wire#w1
      Contact( #Man_Gun_down_2 )
      wire#w3
      Contact( #GUN_DOWN2 )
      P_Trig( #trig[21] )
      S_Coil( #GUN_DOWN2 )
   END_RUNG
   RUNG wire#w3
      I_Contact( #GUN_DOWN2 )
      N_Trig( #trig[22] )
      R_Coil( #GUN_DOWN2 )
   END_RUNG
   RUNG wire#w1
      Contact( #Man_Gun_down_3 )
      wire#w4
      Contact( #GUN_DOWN3 )
      P_Trig( #trig[23] )
      S_Coil( #GUN_DOWN3 )
   END_RUNG
   RUNG wire#w4
      I_Contact( #GUN_DOWN3 )
      N_Trig( #trig[24] )
      R_Coil( #GUN_DOWN3 )
   END_RUNG
   RUNG wire#w1
      Contact( #Man_Gun_down_4 )
      wire#w5
      Contact( #GUN_DOWN4 )
      P_Trig( #trig[25] )
      S_Coil( #GUN_DOWN4 )
   END_RUNG
   RUNG wire#w5
      I_Contact( #GUN_DOWN4 )
      N_Trig( #trig[26] )
      R_Coil( #GUN_DOWN4 )
   END_RUNG
   RUNG wire#w1
      Contact( #Man_Gun_down_5 )
      wire#w6
      Contact( #GUN_DOWN5 )
      P_Trig( #trig[27] )
      S_Coil( #GUN_DOWN5 )
   END_RUNG
   RUNG wire#w6
      I_Contact( #GUN_DOWN5 )
      N_Trig( #trig[28] )
      R_Coil( #GUN_DOWN5 )
   END_RUNG
   RUNG wire#w1
      Contact( #Man_Gun_down_6 )
      wire#w7
      Contact( #GUN_DOWN6 )
      P_Trig( #trig[29] )
      S_Coil( #GUN_DOWN6 )
   END_RUNG
   RUNG wire#w7
      I_Contact( #GUN_DOWN6 )
      N_Trig( #trig[30] )
      R_Coil( #GUN_DOWN6 )
   END_RUNG
   // the same network as SCL:
   #_w1 := #MANUAL OR ("keypad_logic_DB".screen_number = 8);
   #_w2 := #_w1 AND #Man_Gun_down_1;
   #_w3 := #_w2 AND #GUN_DOWN1;
   #_w4 := #_w3 AND NOT #trig[20];   // rising edge
   #trig[20] := #_w3;
   IF #_w4 THEN #GUN_DOWN1 := TRUE; END_IF;
   #_w5 := #_w2 AND NOT #GUN_DOWN1;
   #_w6 := NOT #_w5 AND #trig[21];   // falling edge
   #trig[21] := #_w5;
   IF #_w6 THEN #GUN_DOWN1 := FALSE; END_IF;
   #_w7 := #_w1 AND #Man_Gun_down_2;
   #_w8 := #_w7 AND #GUN_DOWN2;
   #_w9 := #_w8 AND NOT #trig[21];   // rising edge
   #trig[21] := #_w8;
   IF #_w9 THEN #GUN_DOWN2 := TRUE; END_IF;
   #_w10 := #_w7 AND NOT #GUN_DOWN2;
   #_w11 := NOT #_w10 AND #trig[22];   // falling edge
   #trig[22] := #_w10;
   IF #_w11 THEN #GUN_DOWN2 := FALSE; END_IF;
   #_w12 := #_w1 AND #Man_Gun_down_3;
   #_w13 := #_w12 AND #GUN_DOWN3;
   #_w14 := #_w13 AND NOT #trig[23];   // rising edge
   #trig[23] := #_w13;
   IF #_w14 THEN #GUN_DOWN3 := TRUE; END_IF;
   #_w15 := #_w12 AND NOT #GUN_DOWN3;
   #_w16 := NOT #_w15 AND #trig[24];   // falling edge
   #trig[24] := #_w15;
   IF #_w16 THEN #GUN_DOWN3 := FALSE; END_IF;
   #_w17 := #_w1 AND #Man_Gun_down_4;
   #_w18 := #_w17 AND #GUN_DOWN4;
   #_w19 := #_w18 AND NOT #trig[25];   // rising edge
   #trig[25] := #_w18;
   IF #_w19 THEN #GUN_DOWN4 := TRUE; END_IF;
   #_w20 := #_w17 AND NOT #GUN_DOWN4;
   #_w21 := NOT #_w20 AND #trig[26];   // falling edge
   #trig[26] := #_w20;
   IF #_w21 THEN #GUN_DOWN4 := FALSE; END_IF;
   #_w22 := #_w1 AND #Man_Gun_down_5;
   #_w23 := #_w22 AND #GUN_DOWN5;
   #_w24 := #_w23 AND NOT #trig[27];   // rising edge
   #trig[27] := #_w23;
   IF #_w24 THEN #GUN_DOWN5 := TRUE; END_IF;
   #_w25 := #_w22 AND NOT #GUN_DOWN5;
   #_w26 := NOT #_w25 AND #trig[28];   // falling edge
   #trig[28] := #_w25;
   IF #_w26 THEN #GUN_DOWN5 := FALSE; END_IF;
   #_w27 := #_w1 AND #Man_Gun_down_6;
   #_w28 := #_w27 AND #GUN_DOWN6;
   #_w29 := #_w28 AND NOT #trig[29];   // rising edge
   #trig[29] := #_w28;
   IF #_w29 THEN #GUN_DOWN6 := TRUE; END_IF;
   #_w30 := #_w27 AND NOT #GUN_DOWN6;
   #_w31 := NOT #_w30 AND #trig[30];   // falling edge
   #trig[30] := #_w30;
   IF #_w31 THEN #GUN_DOWN6 := FALSE; END_IF;
END_REGION

REGION Network 37
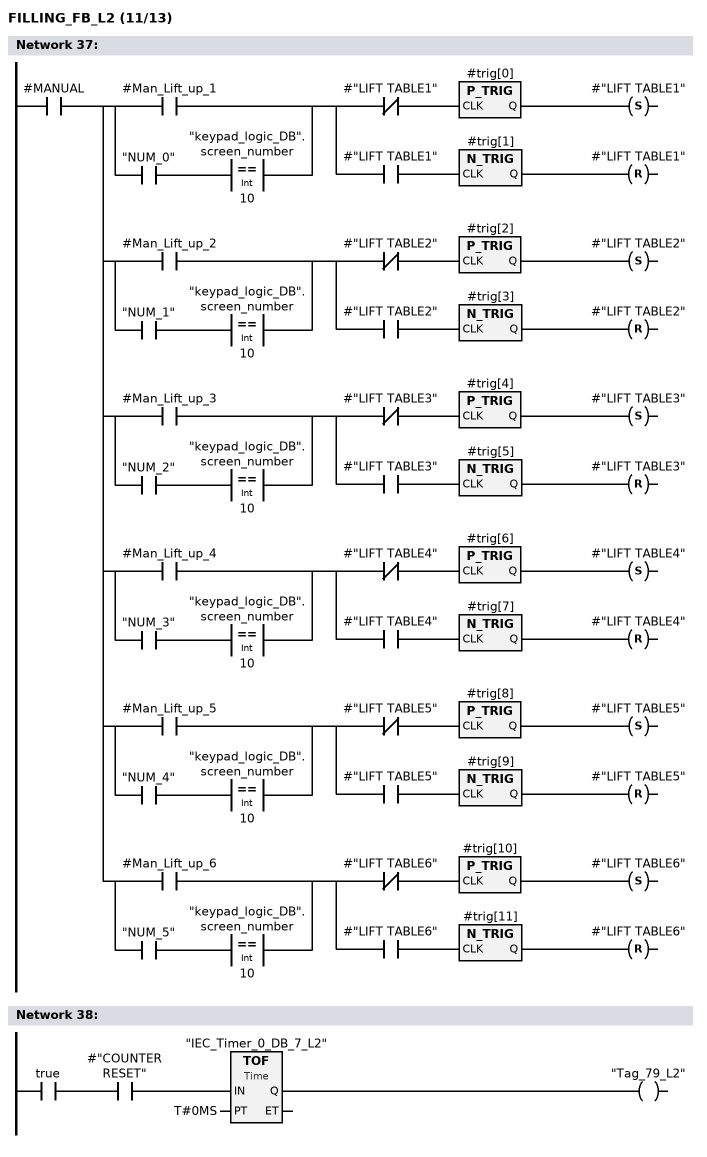
   RUNG wire#powerrail
      Contact( #MANUAL )
      wire#w1
      Contact( #Man_Lift_up_1 )
      wire#w2
      I_Contact( #"LIFT TABLE1" )
      P_Trig( #trig[0] )
      S_Coil( #"LIFT TABLE1" )
   END_RUNG
   RUNG wire#w1
      Contact( "NUM_0" )
      { S7_Templates := "SrcType := Int" } EQ_Contact(in1 := "keypad_logic_DB".screen_number, in2 := 10)
   END_RUNG wire#w2
   RUNG wire#w2
      Contact( #"LIFT TABLE1" )
      N_Trig( #trig[1] )
      R_Coil( #"LIFT TABLE1" )
   END_RUNG
   RUNG wire#w1
      Contact( #Man_Lift_up_2 )
      wire#w3
      I_Contact( #"LIFT TABLE2" )
      P_Trig( #trig[2] )
      S_Coil( #"LIFT TABLE2" )
   END_RUNG
   RUNG wire#w1
      Contact( "NUM_1" )
      { S7_Templates := "SrcType := Int" } EQ_Contact(in1 := "keypad_logic_DB".screen_number, in2 := 10)
   END_RUNG wire#w3
   RUNG wire#w3
      Contact( #"LIFT TABLE2" )
      N_Trig( #trig[3] )
      R_Coil( #"LIFT TABLE2" )
   END_RUNG
   RUNG wire#w1
      Contact( #Man_Lift_up_3 )
      wire#w4
      I_Contact( #"LIFT TABLE3" )
      P_Trig( #trig[4] )
      S_Coil( #"LIFT TABLE3" )
   END_RUNG
   RUNG wire#w1
      Contact( "NUM_2" )
      { S7_Templates := "SrcType := Int" } EQ_Contact(in1 := "keypad_logic_DB".screen_number, in2 := 10)
   END_RUNG wire#w4
   RUNG wire#w4
      Contact( #"LIFT TABLE3" )
      N_Trig( #trig[5] )
      R_Coil( #"LIFT TABLE3" )
   END_RUNG
   RUNG wire#w1
      Contact( #Man_Lift_up_4 )
      wire#w5
      I_Contact( #"LIFT TABLE4" )
      P_Trig( #trig[6] )
      S_Coil( #"LIFT TABLE4" )
   END_RUNG
   RUNG wire#w1
      Contact( "NUM_3" )
      { S7_Templates := "SrcType := Int" } EQ_Contact(in1 := "keypad_logic_DB".screen_number, in2 := 10)
   END_RUNG wire#w5
   RUNG wire#w5
      Contact( #"LIFT TABLE4" )
      N_Trig( #trig[7] )
      R_Coil( #"LIFT TABLE4" )
   END_RUNG
   RUNG wire#w1
      Contact( #Man_Lift_up_5 )
      wire#w6
      I_Contact( #"LIFT TABLE5" )
      P_Trig( #trig[8] )
      S_Coil( #"LIFT TABLE5" )
   END_RUNG
   RUNG wire#w1
      Contact( "NUM_4" )
      { S7_Templates := "SrcType := Int" } EQ_Contact(in1 := "keypad_logic_DB".screen_number, in2 := 10)
   END_RUNG wire#w6
   RUNG wire#w6
      Contact( #"LIFT TABLE5" )
      N_Trig( #trig[9] )
      R_Coil( #"LIFT TABLE5" )
   END_RUNG
   RUNG wire#w1
      Contact( #Man_Lift_up_6 )
      wire#w7
      I_Contact( #"LIFT TABLE6" )
      P_Trig( #trig[10] )
      S_Coil( #"LIFT TABLE6" )
   END_RUNG
   RUNG wire#w1
      Contact( "NUM_5" )
      { S7_Templates := "SrcType := Int" } EQ_Contact(in1 := "keypad_logic_DB".screen_number, in2 := 10)
   END_RUNG wire#w7
   RUNG wire#w7
      Contact( #"LIFT TABLE6" )
      N_Trig( #trig[11] )
      R_Coil( #"LIFT TABLE6" )
   END_RUNG
   // the same network as SCL:
   #_w1 := #MANUAL AND (#Man_Lift_up_1 OR ("NUM_0" AND ("keypad_logic_DB".screen_number = 10)));
   #_w2 := #_w1 AND NOT #"LIFT TABLE1";
   #_w3 := #_w2 AND NOT #trig[0];   // rising edge
   #trig[0] := #_w2;
   IF #_w3 THEN #"LIFT TABLE1" := TRUE; END_IF;
   #_w4 := #_w1 AND #"LIFT TABLE1";
   #_w5 := NOT #_w4 AND #trig[1];   // falling edge
   #trig[1] := #_w4;
   IF #_w5 THEN #"LIFT TABLE1" := FALSE; END_IF;
   #_w6 := #MANUAL AND (#Man_Lift_up_2 OR ("NUM_1" AND ("keypad_logic_DB".screen_number = 10)));
   #_w7 := #_w6 AND NOT #"LIFT TABLE2";
   #_w8 := #_w7 AND NOT #trig[2];   // rising edge
   #trig[2] := #_w7;
   IF #_w8 THEN #"LIFT TABLE2" := TRUE; END_IF;
   #_w9 := #_w6 AND #"LIFT TABLE2";
   #_w10 := NOT #_w9 AND #trig[3];   // falling edge
   #trig[3] := #_w9;
   IF #_w10 THEN #"LIFT TABLE2" := FALSE; END_IF;
   #_w11 := #MANUAL AND (#Man_Lift_up_3 OR ("NUM_2" AND ("keypad_logic_DB".screen_number = 10)));
   #_w12 := #_w11 AND NOT #"LIFT TABLE3";
   #_w13 := #_w12 AND NOT #trig[4];   // rising edge
   #trig[4] := #_w12;
   IF #_w13 THEN #"LIFT TABLE3" := TRUE; END_IF;
   #_w14 := #_w11 AND #"LIFT TABLE3";
   #_w15 := NOT #_w14 AND #trig[5];   // falling edge
   #trig[5] := #_w14;
   IF #_w15 THEN #"LIFT TABLE3" := FALSE; END_IF;
   #_w16 := #MANUAL AND (#Man_Lift_up_4 OR ("NUM_3" AND ("keypad_logic_DB".screen_number = 10)));
   #_w17 := #_w16 AND NOT #"LIFT TABLE4";
   #_w18 := #_w17 AND NOT #trig[6];   // rising edge
   #trig[6] := #_w17;
   IF #_w18 THEN #"LIFT TABLE4" := TRUE; END_IF;
   #_w19 := #_w16 AND #"LIFT TABLE4";
   #_w20 := NOT #_w19 AND #trig[7];   // falling edge
   #trig[7] := #_w19;
   IF #_w20 THEN #"LIFT TABLE4" := FALSE; END_IF;
   #_w21 := #MANUAL AND (#Man_Lift_up_5 OR ("NUM_4" AND ("keypad_logic_DB".screen_number = 10)));
   #_w22 := #_w21 AND NOT #"LIFT TABLE5";
   #_w23 := #_w22 AND NOT #trig[8];   // rising edge
   #trig[8] := #_w22;
   IF #_w23 THEN #"LIFT TABLE5" := TRUE; END_IF;
   #_w24 := #_w21 AND #"LIFT TABLE5";
   #_w25 := NOT #_w24 AND #trig[9];   // falling edge
   #trig[9] := #_w24;
   IF #_w25 THEN #"LIFT TABLE5" := FALSE; END_IF;
   #_w26 := #MANUAL AND (#Man_Lift_up_6 OR ("NUM_5" AND ("keypad_logic_DB".screen_number = 10)));
   #_w27 := #_w26 AND NOT #"LIFT TABLE6";
   #_w28 := #_w27 AND NOT #trig[10];   // rising edge
   #trig[10] := #_w27;
   IF #_w28 THEN #"LIFT TABLE6" := TRUE; END_IF;
   #_w29 := #_w26 AND #"LIFT TABLE6";
   #_w30 := NOT #_w29 AND #trig[11];   // falling edge
   #trig[11] := #_w29;
   IF #_w30 THEN #"LIFT TABLE6" := FALSE; END_IF;
END_REGION

REGION Network 38
   RUNG wire#powerrail
      Contact( true )
      Contact( #"COUNTER RESET" )
      { S7_Templates := "time_type := Time" } "IEC_Timer_0_DB_7_L2".TOF(pt := T#0MS, et =>)
      Coil( "Tag_79_L2" )
   END_RUNG
   // the same network as SCL:
   "IEC_Timer_0_DB_7_L2".TOF(IN := true AND #"COUNTER RESET", PT := T#0MS);
   "Tag_79_L2" := "IEC_Timer_0_DB_7_L2".Q;
END_REGION

REGION Network 39
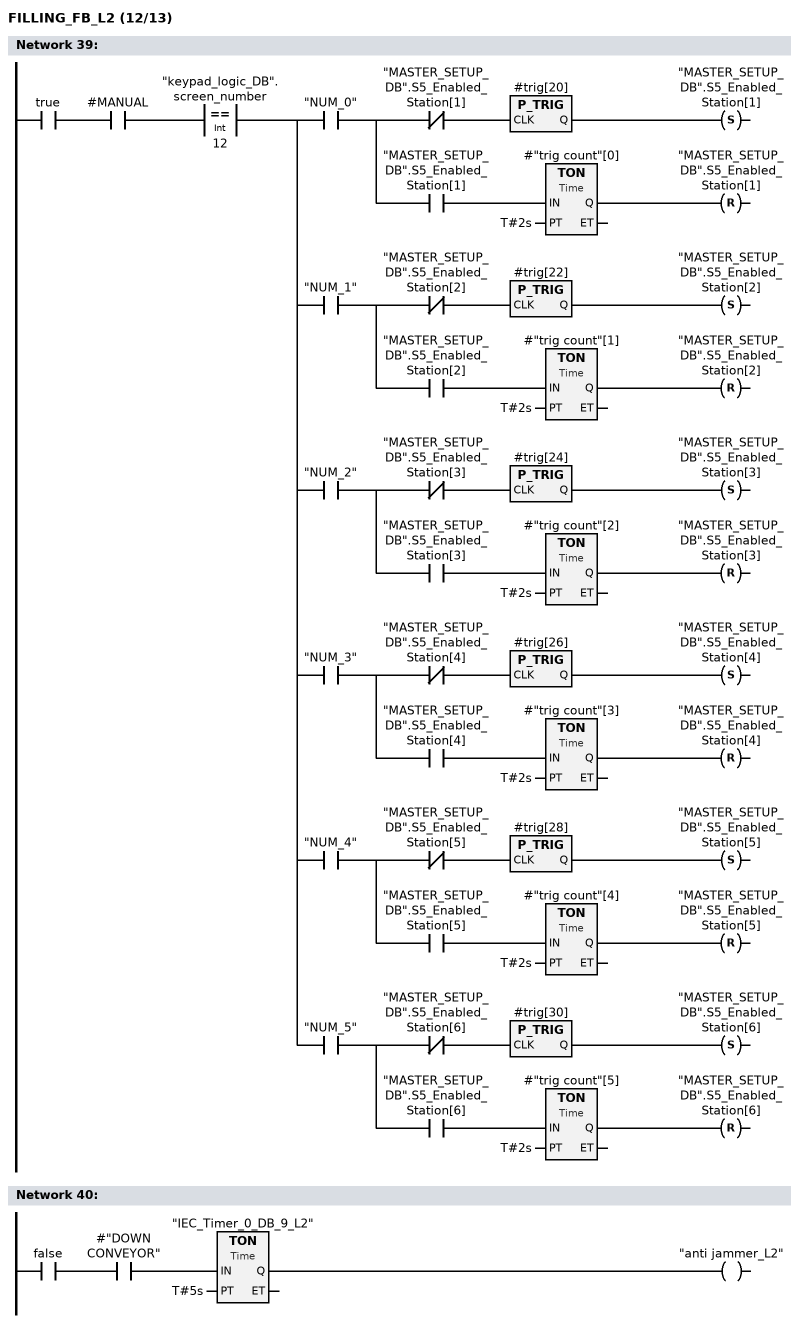
   RUNG wire#powerrail
      Contact( true )
      Contact( #MANUAL )
      { S7_Templates := "SrcType := Int" } EQ_Contact(in1 := "keypad_logic_DB".screen_number, in2 := 12)
      wire#w1
      Contact( "NUM_0" )
      wire#w2
      I_Contact( "MASTER_SETUP_DB".S5_Enabled_Station[1] )
      P_Trig( #trig[20] )
      S_Coil( "MASTER_SETUP_DB".S5_Enabled_Station[1] )
   END_RUNG
   RUNG wire#w2
      Contact( "MASTER_SETUP_DB".S5_Enabled_Station[1] )
      { S7_Templates := "time_type := Time" } #"trig count"[0].TON(pt := T#2s, et =>)
      R_Coil( "MASTER_SETUP_DB".S5_Enabled_Station[1] )
   END_RUNG
   RUNG wire#w1
      Contact( "NUM_1" )
      wire#w3
      I_Contact( "MASTER_SETUP_DB".S5_Enabled_Station[2] )
      P_Trig( #trig[22] )
      S_Coil( "MASTER_SETUP_DB".S5_Enabled_Station[2] )
   END_RUNG
   RUNG wire#w3
      Contact( "MASTER_SETUP_DB".S5_Enabled_Station[2] )
      { S7_Templates := "time_type := Time" } #"trig count"[1].TON(pt := T#2s, et =>)
      R_Coil( "MASTER_SETUP_DB".S5_Enabled_Station[2] )
   END_RUNG
   RUNG wire#w1
      Contact( "NUM_2" )
      wire#w4
      I_Contact( "MASTER_SETUP_DB".S5_Enabled_Station[3] )
      P_Trig( #trig[24] )
      S_Coil( "MASTER_SETUP_DB".S5_Enabled_Station[3] )
   END_RUNG
   RUNG wire#w4
      Contact( "MASTER_SETUP_DB".S5_Enabled_Station[3] )
      { S7_Templates := "time_type := Time" } #"trig count"[2].TON(pt := T#2s, et =>)
      R_Coil( "MASTER_SETUP_DB".S5_Enabled_Station[3] )
   END_RUNG
   RUNG wire#w1
      Contact( "NUM_3" )
      wire#w5
      I_Contact( "MASTER_SETUP_DB".S5_Enabled_Station[4] )
      P_Trig( #trig[26] )
      S_Coil( "MASTER_SETUP_DB".S5_Enabled_Station[4] )
   END_RUNG
   RUNG wire#w5
      Contact( "MASTER_SETUP_DB".S5_Enabled_Station[4] )
      { S7_Templates := "time_type := Time" } #"trig count"[3].TON(pt := T#2s, et =>)
      R_Coil( "MASTER_SETUP_DB".S5_Enabled_Station[4] )
   END_RUNG
   RUNG wire#w1
      Contact( "NUM_4" )
      wire#w6
      I_Contact( "MASTER_SETUP_DB".S5_Enabled_Station[5] )
      P_Trig( #trig[28] )
      S_Coil( "MASTER_SETUP_DB".S5_Enabled_Station[5] )
   END_RUNG
   RUNG wire#w6
      Contact( "MASTER_SETUP_DB".S5_Enabled_Station[5] )
      { S7_Templates := "time_type := Time" } #"trig count"[4].TON(pt := T#2s, et =>)
      R_Coil( "MASTER_SETUP_DB".S5_Enabled_Station[5] )
   END_RUNG
   RUNG wire#w1
      Contact( "NUM_5" )
      wire#w7
      I_Contact( "MASTER_SETUP_DB".S5_Enabled_Station[6] )
      P_Trig( #trig[30] )
      S_Coil( "MASTER_SETUP_DB".S5_Enabled_Station[6] )
   END_RUNG
   RUNG wire#w7
      Contact( "MASTER_SETUP_DB".S5_Enabled_Station[6] )
      { S7_Templates := "time_type := Time" } #"trig count"[5].TON(pt := T#2s, et =>)
      R_Coil( "MASTER_SETUP_DB".S5_Enabled_Station[6] )
   END_RUNG
   // the same network as SCL:
   #_w1 := true AND #MANUAL AND ("keypad_logic_DB".screen_number = 12);
   #_w2 := #_w1 AND "NUM_0";
   #_w3 := #_w2 AND NOT "MASTER_SETUP_DB".S5_Enabled_Station[1];
   #_w4 := #_w3 AND NOT #trig[20];   // rising edge
   #trig[20] := #_w3;
   IF #_w4 THEN "MASTER_SETUP_DB".S5_Enabled_Station[1] := TRUE; END_IF;
   #"trig count"[0].TON(IN := #_w2 AND "MASTER_SETUP_DB".S5_Enabled_Station[1], PT := T#2s);
   IF #"trig count"[0].Q THEN "MASTER_SETUP_DB".S5_Enabled_Station[1] := FALSE; END_IF;
   #_w5 := #_w1 AND "NUM_1";
   #_w6 := #_w5 AND NOT "MASTER_SETUP_DB".S5_Enabled_Station[2];
   #_w7 := #_w6 AND NOT #trig[22];   // rising edge
   #trig[22] := #_w6;
   IF #_w7 THEN "MASTER_SETUP_DB".S5_Enabled_Station[2] := TRUE; END_IF;
   #"trig count"[1].TON(IN := #_w5 AND "MASTER_SETUP_DB".S5_Enabled_Station[2], PT := T#2s);
   IF #"trig count"[1].Q THEN "MASTER_SETUP_DB".S5_Enabled_Station[2] := FALSE; END_IF;
   #_w8 := #_w1 AND "NUM_2";
   #_w9 := #_w8 AND NOT "MASTER_SETUP_DB".S5_Enabled_Station[3];
   #_w10 := #_w9 AND NOT #trig[24];   // rising edge
   #trig[24] := #_w9;
   IF #_w10 THEN "MASTER_SETUP_DB".S5_Enabled_Station[3] := TRUE; END_IF;
   #"trig count"[2].TON(IN := #_w8 AND "MASTER_SETUP_DB".S5_Enabled_Station[3], PT := T#2s);
   IF #"trig count"[2].Q THEN "MASTER_SETUP_DB".S5_Enabled_Station[3] := FALSE; END_IF;
   #_w11 := #_w1 AND "NUM_3";
   #_w12 := #_w11 AND NOT "MASTER_SETUP_DB".S5_Enabled_Station[4];
   #_w13 := #_w12 AND NOT #trig[26];   // rising edge
   #trig[26] := #_w12;
   IF #_w13 THEN "MASTER_SETUP_DB".S5_Enabled_Station[4] := TRUE; END_IF;
   #"trig count"[3].TON(IN := #_w11 AND "MASTER_SETUP_DB".S5_Enabled_Station[4], PT := T#2s);
   IF #"trig count"[3].Q THEN "MASTER_SETUP_DB".S5_Enabled_Station[4] := FALSE; END_IF;
   #_w14 := #_w1 AND "NUM_4";
   #_w15 := #_w14 AND NOT "MASTER_SETUP_DB".S5_Enabled_Station[5];
   #_w16 := #_w15 AND NOT #trig[28];   // rising edge
   #trig[28] := #_w15;
   IF #_w16 THEN "MASTER_SETUP_DB".S5_Enabled_Station[5] := TRUE; END_IF;
   #"trig count"[4].TON(IN := #_w14 AND "MASTER_SETUP_DB".S5_Enabled_Station[5], PT := T#2s);
   IF #"trig count"[4].Q THEN "MASTER_SETUP_DB".S5_Enabled_Station[5] := FALSE; END_IF;
   #_w17 := #_w1 AND "NUM_5";
   #_w18 := #_w17 AND NOT "MASTER_SETUP_DB".S5_Enabled_Station[6];
   #_w19 := #_w18 AND NOT #trig[30];   // rising edge
   #trig[30] := #_w18;
   IF #_w19 THEN "MASTER_SETUP_DB".S5_Enabled_Station[6] := TRUE; END_IF;
   #"trig count"[5].TON(IN := #_w17 AND "MASTER_SETUP_DB".S5_Enabled_Station[6], PT := T#2s);
   IF #"trig count"[5].Q THEN "MASTER_SETUP_DB".S5_Enabled_Station[6] := FALSE; END_IF;
END_REGION

REGION Network 40
   RUNG wire#powerrail
      Contact( false )
      Contact( #"DOWN CONVEYOR" )
      { S7_Templates := "time_type := Time" } "IEC_Timer_0_DB_9_L2".TON(pt := T#5s, et =>)
      Coil( "anti jammer_L2" )
   END_RUNG
   // the same network as SCL:
   "IEC_Timer_0_DB_9_L2".TON(IN := false AND #"DOWN CONVEYOR", PT := T#5s);
   "anti jammer_L2" := "IEC_Timer_0_DB_9_L2".Q;
END_REGION

REGION Network 41
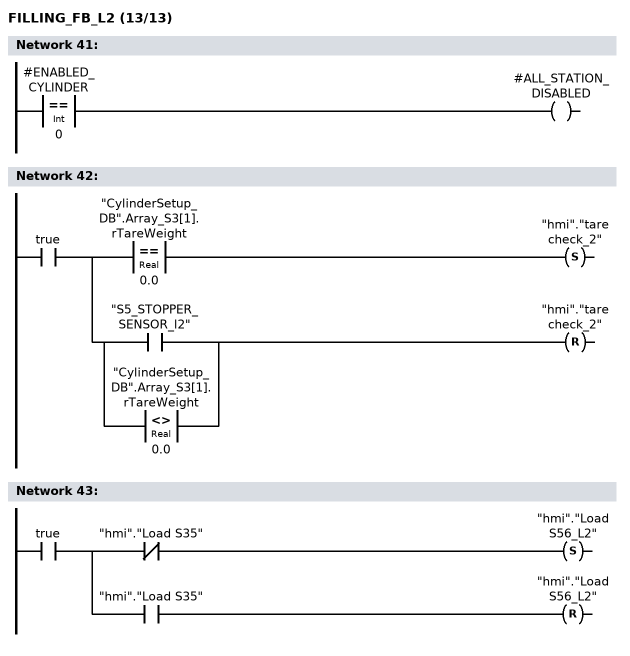
   RUNG wire#powerrail
      { S7_Templates := "SrcType := Int" } EQ_Contact(in1 := #ENABLED_CYLINDER, in2 := 0)
      Coil( #ALL_STATION_DISABLED )
   END_RUNG
   // the same network as SCL:
   #ALL_STATION_DISABLED := #ENABLED_CYLINDER = 0;
END_REGION

REGION Network 42
   RUNG wire#powerrail
      Contact( true )
      wire#w1
      { S7_Templates := "SrcType := Real" } EQ_Contact(in1 := "CylinderSetup_DB".Array_S3[1].rTareWeight, in2 := 0.0)
      S_Coil( "hmi"."tare check_2" )
   END_RUNG
   RUNG wire#w1
      Contact( "S5_STOPPER_SENSOR_l2" )
      wire#w2
      R_Coil( "hmi"."tare check_2" )
   END_RUNG
   RUNG wire#w1
      { S7_Templates := "SrcType := Real" } NE_Contact(in1 := "CylinderSetup_DB".Array_S3[1].rTareWeight, in2 := 0.0)
   END_RUNG wire#w2
   // the same network as SCL:
   IF true AND ("CylinderSetup_DB".Array_S3[1].rTareWeight = 0.0) THEN "hmi"."tare check_2" := TRUE; END_IF;
   IF true AND ("S5_STOPPER_SENSOR_l2" OR ("CylinderSetup_DB".Array_S3[1].rTareWeight <> 0.0)) THEN
       "hmi"."tare check_2" := FALSE;
   END_IF;
END_REGION

REGION Network 43
   RUNG wire#powerrail
      Contact( true )
      wire#w1
      I_Contact( "hmi"."Load S35" )
      S_Coil( "hmi"."Load S56_L2" )
   END_RUNG
   RUNG wire#w1
      Contact( "hmi"."Load S35" )
      R_Coil( "hmi"."Load S56_L2" )
   END_RUNG
   // the same network as SCL:
   IF true AND NOT "hmi"."Load S35" THEN "hmi"."Load S56_L2" := TRUE; END_IF;
   IF true AND "hmi"."Load S35" THEN "hmi"."Load S56_L2" := FALSE; END_IF;
END_REGION
END_FUNCTION_BLOCK
